(*!
<summary>Checks concrete metadata and name stability across cancellation and Reset for all sixteen tasks.</summary>
<description>Each concrete reset hook is exercised. Cancellation occurs before issuing a native request.</description>
*)
METHOD PROTECTED ExecuteTest
VAR
	expectedTypes : ARRAY [0..15] OF STRING(80) := [
		'CheckDirectoryExists',
		'CreateDirectory',
		'CreateDirectoryIfNotExists',
		'RemoveEmptyDirectory',
		'RemoveEmptyDirectoryIfExists',
		'DeleteFile',
		'RenameFile',
		'LoadFile',
		'FileContentManager',
		'CheckEndOfFile',
		'GetPositionInFile',
		'SetPositionInFile',
		'ReadBytesFromFile',
		'ReadString255FromFile',
		'WriteBytesToFile',
		'WriteString255ToFile'
	];
	expectedName : WSTRING;
	i : DINT;
	caseName : WSTRING;
	started : BOOL;
	cancelled : BOOL;
END_VAR
FOR i := LOWER_BOUND(_Tasks, 1) TO UPPER_BOUND(_Tasks, 1) DO
	caseName := TO_WSTRING(expectedTypes[i]);
	expectedName := TO_WSTRING(TOF_Core.Strings.Concat255(
		expectedTypes[i],
		' (0x',
		Tc2_Utilities.LWORD_TO_HEXSTR(in := TO_LWORD(_Tasks[i].SelfAddress), iPrecision := 16, bLoCase := FALSE),
		')'
	));
	Assert.ThatBool(
		actual := _Tasks[i].Name = expectedName,
		message := TOF_Core.WideStrings.Concat255(caseName, ": Default name must include the concrete type and address")
	).IsTrue();
	Assert.ThatBool(
		actual := _Tasks[i].ClassName = expectedTypes[i],
		message := TOF_Core.WideStrings.Concat255(caseName, ": ", "ClassName must identify the concrete task")
	).IsTrue();
	Assert.ThatBool(
		actual := _Tasks[i].NamespaceName = 'TOF_FileSystem',
		message := TOF_Core.WideStrings.Concat255(caseName, ": ", "Task namespace must identify FileSystem")
	).IsTrue();
	Assert.ThatBool(
		actual := _Tasks[i].State.Ready,
		message := TOF_Core.WideStrings.Concat255(caseName, ": Metadata must leave the task READY")
	).IsTrue();
	started := _Tasks[i].Start();
	Assert.ThatBool(
		actual := started,
		message := TOF_Core.WideStrings.Concat255(caseName, ": ", "Task must accept Start before cancellation")
	).IsTrue();

	IF NOT started THEN
		CONTINUE;
	END_IF

	cancelled := _Tasks[i].Cancel();
	Assert.ThatBool(
		actual := cancelled,
		message := TOF_Core.WideStrings.Concat255(caseName, ": ", "Task must accept Cancel before Execute")
	).IsTrue();

	IF NOT cancelled THEN
		CONTINUE;
	END_IF

	_Tasks[i].Execute();
	Assert.ThatBool(
		actual := _Tasks[i].State.Stopped,
		message := TOF_Core.WideStrings.Concat255(caseName, ": ", "Task must stop after cancellation")
	).IsTrue();
	Assert.ThatBool(
		actual := _Tasks[i].FinalStopReason.ExternalCancel,
		message := TOF_Core.WideStrings.Concat255(caseName, ": ", "Pre-submission cancellation must retain its reason")
	).IsTrue();
	Assert.ThatBool(
		actual := _Tasks[i].Reset(),
		message := TOF_Core.WideStrings.Concat255(caseName, ": ", "Stopped task must accept Reset")
	).IsTrue();
	Assert.ThatBool(
		actual := _Tasks[i].State.Ready,
		message := TOF_Core.WideStrings.Concat255(caseName, ": Reset must restore READY")
	).IsTrue();
	Assert.ThatBool(
		actual := _Tasks[i].Name = expectedName,
		message := TOF_Core.WideStrings.Concat255(caseName, ": Reset must preserve the stored default name")
	).IsTrue();
END_FOR

Assert.ThatBool(
	actual := _ExplicitDirectory.Name = "Explicit directory",
	message := "Directory explicit name must be copied"
).IsTrue();
Assert.ThatBool(
	actual := _ExplicitManager.Name = "Explicit manager",
	message := "Manager explicit name must be copied"
).IsTrue();
Assert.ThatBool(
	actual := _ExplicitRead.Name = "Explicit read",
	message := "Content task explicit name must be copied"
).IsTrue();
END_METHOD

(*!
<summary>Restores the fixtures after a completed or interrupted test.</summary>
<description>
Advances a running task only after cancellation is recorded. Resets fixtures only when they are not already READY.
</description>
*)
METHOD PROTECTED AfterTest
VAR
	i : DINT;
END_VAR
FOR i := LOWER_BOUND(_Tasks, 1) TO UPPER_BOUND(_Tasks, 1) DO
	IF _Tasks[i].State.Running THEN
		IF _Tasks[i].OriginalStopReason.ExternalCancel OR_ELSE _Tasks[i].Cancel() THEN
			_Tasks[i].Execute();
		END_IF
	END_IF

	IF NOT _Tasks[i].State.Ready THEN
		Assert.ThatBool(
			actual := _Tasks[i].Reset(),
			message := TOF_Core.WideStrings.Concat255(_Tasks[i].Name, " must accept Reset during cleanup")
		).IsTrue();
	END_IF
END_FOR
END_METHOD

//! <summary>Borrows the concrete class name for the lifetime of this instance; callers must not modify it.</summary>
{attribute 'monitoring' := 'call'}
PROPERTY ClassName : REFERENCE TO STRING
GET
ClassName REF= _ClassName;
END_GET
END_PROPERTY

//! <summary>Borrows the compiler-initialized namespace; callers must not modify the returned reference.</summary>
{attribute 'monitoring' := 'call'}
PROPERTY NamespaceName : REFERENCE TO STRING
GET
NamespaceName REF= CurrentNamespace.Name;
END_GET
END_PROPERTY

//! <summary>Reports the complete concrete instance size, excluding separately allocated storage.</summary>
{attribute 'monitoring' := 'call'}
PROPERTY SelfSize : ULINT
GET
SelfSize := XSIZEOF(THIS^);
END_GET
END_PROPERTY

END_FUNCTION_BLOCK

// ---- Tests/Files/FileSystemUnboundContentTest.TcPOU
(*
SPDX-FileCopyrightText: © 2026 Oleksandr Tiutyk <trofimich@gmail.com>
SPDX-License-Identifier: MIT
License: https://opensource.org/license/mit
*)

(*!
<summary>Checks all seven unbound content operations and their guarded failure/reset results.</summary>
<description>
The fixture belongs to the runner task and is kept between runs. The test drives no native file requests.
</description>
*)

{attribute 'no_assign'}
{attribute 'no_explicit_call' := 'do not call this function block directly'}
FUNCTION_BLOCK FileSystemUnboundContentTest EXTENDS TOF_Testing.SingleCycleTest
VAR_STAT
	{attribute 'hide'}
	_ClassName : STRING := __POUNAME();
END_VAR
VAR
	_CheckEof : TOF_FileSystem.CheckEndOfFile(name := "unbound CheckEndOfFile");
	_GetPosition : TOF_FileSystem.GetPositionInFile(name := "unbound GetPositionInFile");
	_SetPosition : TOF_FileSystem.SetPositionInFile(name := "unbound SetPositionInFile");
	_ReadBytes : TOF_FileSystem.ReadBytesFromFile(name := "unbound ReadBytesFromFile");
	_ReadString : TOF_FileSystem.ReadString255FromFile(name := "unbound ReadString255FromFile");
	_WriteBytes : TOF_FileSystem.WriteBytesToFile(name := "unbound WriteBytesToFile");
	_WriteString : TOF_FileSystem.WriteString255ToFile(name := "unbound WriteString255ToFile");

	_Tasks : ARRAY [0..6] OF TOF_Tasks.ITask :=
	[
		_CheckEof,
		_GetPosition,
		_SetPosition,
		_ReadBytes,
		_ReadString,
		_WriteBytes,
		_WriteString
	];
END_VAR

(*!
<summary>Checks all seven unbound content operations and their guarded failure/reset results.</summary>
<description>Requires the missing-member diagnostic and checks guarded results in each lifecycle phase.</description>
*)
METHOD PROTECTED ExecuteTest
VAR
	i : DINT;
	message : STRING(255);
	caseName : WSTRING;
	started : BOOL;
END_VAR
checkGuardedResults(phase := "Before Start");

FOR i := LOWER_BOUND(_Tasks, 1) TO UPPER_BOUND(_Tasks, 1) DO
	caseName := _Tasks[i].Name;
	started := _Tasks[i].Start();
	Assert.ThatBool(
		actual := started,
		message := TOF_Core.WideStrings.Concat255(caseName, ": ", "Start must precede validation")
	).IsTrue();

	IF NOT started THEN
		CONTINUE;
	END_IF

	_Tasks[i].Execute();
	_Tasks[i].Execute();
	Assert.ThatBool(
		actual := _Tasks[i].State.Stopped,
		message := TOF_Core.WideStrings.Concat255(caseName, ": ", "Unbound operation must finish failure cleanup")
	).IsTrue();
	Assert.ThatBool(
		actual := _Tasks[i].FinalStopReason.Failure,
		message := TOF_Core.WideStrings.Concat255(caseName, ": ", "Unbound operation must fail")
	).IsTrue();
	message := TO_STRING(_Tasks[i].FinalStopReason.Message);
	Assert.ThatBool(
		actual := TOF_Core.Strings.Contains(
			stringToSearchIn := message,
			stringToFind := '$27FileHandleResource$27'
		),
		message := TOF_Core.WideStrings.Concat255(caseName, ": ", "Unbound failure must identify the missing resource")
	).IsTrue();
END_FOR

checkGuardedResults(phase := "After failure");

FOR i := LOWER_BOUND(_Tasks, 1) TO UPPER_BOUND(_Tasks, 1) DO
	Assert.ThatBool(
		actual := _Tasks[i].Reset(),
		message := TOF_Core.WideStrings.Concat255(_Tasks[i].Name, " must accept Reset")
	).IsTrue();
	Assert.ThatBool(
		actual := _Tasks[i].State.Ready,
		message := TOF_Core.WideStrings.Concat255(_Tasks[i].Name, " must return to READY")
	).IsTrue();
END_FOR

checkGuardedResults(phase := "After Reset");
END_METHOD

(*!
<summary>Checks result defaults when no successful file operation is available.</summary>
<param name="phase">Identifies the observed lifecycle phase in assertion messages.</param>
*)
METHOD PRIVATE checkGuardedResults
VAR_INPUT
	phase : WSTRING;
END_VAR
Assert.ThatBool(
	actual := _CheckEof.IsEndOfFile,
	message := TOF_Core.WideStrings.Concat255(phase, ": CheckEndOfFile.IsEndOfFile")
).IsFalse();
Assert.ThatBool(
	actual := _GetPosition.Position = TOF_Core.SignedInt32.ZERO,
	message := TOF_Core.WideStrings.Concat255(phase, ": ", "Unsuccessful tell must expose zero")
).IsTrue();
Assert.ThatBool(
	actual := _ReadBytes.ActuallyReadBytes = TOF_Core.UnsignedInt32.ZERO,
	message := TOF_Core.WideStrings.Concat255(phase, ": ", "Unsuccessful read count must be zero")
).IsTrue();
Assert.ThatBool(
	actual := _ReadBytes.IsEndOfFile,
	message := TOF_Core.WideStrings.Concat255(phase, ": ", "Unsuccessful read must not expose EOF")
).IsFalse();
Assert.ThatBool(
	actual := _ReadString.ReadString = '',
	message := TOF_Core.WideStrings.Concat255(phase, ": ", "Unsuccessful string read must expose an empty buffer")
).IsTrue();
Assert.ThatBool(
	actual := _ReadString.IsEndOfFile,
	message := TOF_Core.WideStrings.Concat255(phase, ": ", "Unsuccessful string read must not expose EOF")
).IsFalse();
Assert.ThatBool(
	actual := _WriteBytes.ActuallyWrittenBytes = TOF_Core.UnsignedInt32.ZERO,
	message := TOF_Core.WideStrings.Concat255(phase, ": ", "Unsuccessful write count must be zero")
).IsTrue();
END_METHOD

(*!
<summary>Restores the fixtures after a completed or interrupted test.</summary>
<description>
Advances a running task only after cancellation is recorded. Resets fixtures only when they are not already READY.
</description>
*)
METHOD PROTECTED AfterTest
VAR
	i : DINT;
END_VAR
FOR i := LOWER_BOUND(_Tasks, 1) TO UPPER_BOUND(_Tasks, 1) DO
	IF _Tasks[i].State.Running THEN
		IF _Tasks[i].OriginalStopReason.ExternalCancel OR_ELSE _Tasks[i].Cancel() THEN
			_Tasks[i].Execute();
		END_IF
	END_IF

	IF NOT _Tasks[i].State.Ready THEN
		Assert.ThatBool(
			actual := _Tasks[i].Reset(),
			message := TOF_Core.WideStrings.Concat255(_Tasks[i].Name, " must accept Reset during cleanup")
		).IsTrue();
	END_IF
END_FOR
END_METHOD

//! <summary>Borrows the concrete class name for the lifetime of this instance; callers must not modify it.</summary>
{attribute 'monitoring' := 'call'}
PROPERTY ClassName : REFERENCE TO STRING
GET
ClassName REF= _ClassName;
END_GET
END_PROPERTY

//! <summary>Borrows the compiler-initialized namespace; callers must not modify the returned reference.</summary>
{attribute 'monitoring' := 'call'}
PROPERTY NamespaceName : REFERENCE TO STRING
GET
NamespaceName REF= CurrentNamespace.Name;
END_GET
END_PROPERTY

//! <summary>Reports the complete concrete instance size, excluding separately allocated storage.</summary>
{attribute 'monitoring' := 'call'}
PROPERTY SelfSize : ULINT
GET
SelfSize := XSIZEOF(THIS^);
END_GET
END_PROPERTY

END_FUNCTION_BLOCK

// ---- Tests/Files/FileSystemLoadBufferTest.TcPOU
(*
SPDX-FileCopyrightText: © 2026 Oleksandr Tiutyk <trofimich@gmail.com>
SPDX-License-Identifier: MIT
License: https://opensource.org/license/mit
*)

(*!
<summary>Checks null/zero load buffers and the corrected TargetBufferSize diagnostic without native I/O.</summary>
<description>
The fixture belongs to the runner task and is kept between runs. The test drives no native file requests.
</description>
*)

{attribute 'no_assign'}
{attribute 'no_explicit_call' := 'do not call this function block directly'}
FUNCTION_BLOCK FileSystemLoadBufferTest EXTENDS TOF_Testing.SingleCycleTest
VAR_STAT
	{attribute 'hide'}
	_ClassName : STRING := __POUNAME();
END_VAR
VAR
	_Load : TOF_FileSystem.LoadFile(name := "load preconditions");
	_Buffer : BYTE;
END_VAR

(*!
<summary>Checks null/zero load buffers and the corrected TargetBufferSize diagnostic without native I/O.</summary>
<description>Checks the buffer guard order and confirms the fixture can be reconfigured before native submission.</description>
*)
METHOD PROTECTED ExecuteTest
VAR
	started : BOOL;
	cancelled : BOOL;
END_VAR
_Buffer := BYTE#16#A5;
_Load.FilePath := 'unused.bin';

IF NOT checkInvalidBuffer(
	targetBuffer := TOF_Core.Memory.NULL_ADDRESS,
	size := 1,
	propertyToken := '$27TargetBuffer$27',
	caseName := "Null buffer"
)
	OR_ELSE NOT checkInvalidBuffer(
		targetBuffer := ADR(_Buffer),
		size := TOF_Core.UnsignedInt32.ZERO,
		propertyToken := '$27TargetBufferSize$27',
		caseName := "Zero buffer size"
	)
	OR_ELSE NOT checkInvalidBuffer(
		targetBuffer := TOF_Core.Memory.NULL_ADDRESS,
		size := TOF_Core.UnsignedInt32.ZERO,
		propertyToken := '$27TargetBuffer$27',
		caseName := "Null buffer and zero size"
	)
THEN
	RETURN;
END_IF

_Load.TargetBuffer := ADR(_Buffer);
_Load.TargetBufferSize := 1;
started := _Load.Start();
Assert.ThatBool(actual := started, message := "Reconfigured load must accept Start").IsTrue();

IF NOT started THEN
	RETURN;
END_IF

cancelled := _Load.Cancel();
Assert.ThatBool(actual := cancelled, message := "Reconfigured load must accept pre-submission cancellation").IsTrue();

IF NOT cancelled THEN
	RETURN;
END_IF

_Load.Execute();
Assert.ThatBool(actual := _Load.State.Stopped, message := "Cancelled load must stop before submission").IsTrue();
Assert.ThatBool(
	actual := _Load.FinalStopReason.ExternalCancel,
	message := "Pre-submission load cancellation must preserve its reason"
).IsTrue();
Assert.ThatUDInt(actual := _Load.LoadedBytesCount, message := "Cancelled load byte count").ToBe(
	expected := TOF_Core.UnsignedInt32.ZERO
);
Assert.ThatByte(actual := _Buffer, message := "Cancelled load must preserve the caller buffer").ToBe(
	expected := BYTE#16#A5
);
END_METHOD

(*!
<summary>Checks one invalid buffer configuration and resets the stopped task.</summary>
<description>
The reason must identify the exact rejected member before any native request. The caller buffer keeps its sentinel.
Returns TRUE only after the task has accepted Reset and is READY for the next configuration.
</description>
<param name="targetBuffer">Buffer address to pass to LoadFile.</param>
<param name="size">Configured buffer size in bytes.</param>
<param name="propertyToken">Expected member name including the diagnostic quotes.</param>
<param name="caseName">Identifies the buffer configuration in the assertion messages.</param>
*)
METHOD PRIVATE checkInvalidBuffer : BOOL
VAR_INPUT
	targetBuffer : POINTER TO BYTE;
	size : UDINT;
	propertyToken : STRING(32);
	caseName : WSTRING;
END_VAR
VAR
	started : BOOL;
	message : STRING(255);
	resetAccepted : BOOL;
END_VAR
_Load.TargetBuffer := targetBuffer;
_Load.TargetBufferSize := size;
started := _Load.Start();
Assert.ThatBool(
	actual := started,
	message := TOF_Core.WideStrings.Concat255(caseName, ": Start must precede buffer validation")
).IsTrue();

IF NOT started THEN
	RETURN;
END_IF

_Load.Execute();
_Load.Execute();
Assert.ThatBool(
	actual := _Load.State.Stopped,
	message := TOF_Core.WideStrings.Concat255(caseName, ": must finish stopping")
).IsTrue();
Assert.ThatBool(
	actual := _Load.FinalStopReason.Failure,
	message := TOF_Core.WideStrings.Concat255(caseName, ": must fail")
).IsTrue();
message := TO_STRING(_Load.FinalStopReason.Message);
Assert.ThatBool(
	actual := TOF_Core.Strings.Contains(stringToSearchIn := message, stringToFind := propertyToken),
	message := TOF_Core.WideStrings.Concat255(caseName, ": expected diagnostic for ", TO_WSTRING(propertyToken))
).IsTrue();
Assert.ThatUDInt(
	actual := _Load.LoadedBytesCount,
	message := TOF_Core.WideStrings.Concat255(caseName, ": loaded byte count")
).ToBe(expected := TOF_Core.UnsignedInt32.ZERO);
Assert.ThatByte(
	actual := _Buffer,
	message := TOF_Core.WideStrings.Concat255(caseName, ": caller buffer sentinel")
).ToBe(expected := BYTE#16#A5);

resetAccepted := _Load.Reset();
Assert.ThatBool(
	actual := resetAccepted,
	message := TOF_Core.WideStrings.Concat255(caseName, ": must accept Reset")
).IsTrue();
Assert.ThatBool(
	actual := _Load.State.Ready,
	message := TOF_Core.WideStrings.Concat255(caseName, ": Reset must restore READY")
).IsTrue();
checkInvalidBuffer := resetAccepted AND_THEN _Load.State.Ready;
END_METHOD

(*!
<summary>Resets the load task after cancellation, including after an interrupted assertion sequence.</summary>
<description>
Advances a running task only on its cancellation path and reports a task that cannot be reset.
</description>
*)
METHOD PROTECTED AfterTest
IF _Load.State.Running THEN
	IF _Load.OriginalStopReason.ExternalCancel OR_ELSE _Load.Cancel() THEN
		_Load.Execute();
	END_IF
END_IF

Assert.ThatBool(
	actual := _Load.Reset(),
	message := "Load task must be ready after cleanup"
).IsTrue();
END_METHOD

//! <summary>Borrows the concrete class name for the lifetime of this instance; callers must not modify it.</summary>
{attribute 'monitoring' := 'call'}
PROPERTY ClassName : REFERENCE TO STRING
GET
ClassName REF= _ClassName;
END_GET
END_PROPERTY

//! <summary>Borrows the compiler-initialized namespace; callers must not modify the returned reference.</summary>
{attribute 'monitoring' := 'call'}
PROPERTY NamespaceName : REFERENCE TO STRING
GET
NamespaceName REF= CurrentNamespace.Name;
END_GET
END_PROPERTY

//! <summary>Reports the complete concrete instance size, excluding separately allocated storage.</summary>
{attribute 'monitoring' := 'call'}
PROPERTY SelfSize : ULINT
GET
SelfSize := XSIZEOF(THIS^);
END_GET
END_PROPERTY

END_FUNCTION_BLOCK

// ---- Tests/Files/FileSystemQueueBindingTest.TcPOU
(*
SPDX-FileCopyrightText: © 2026 Oleksandr Tiutyk <trofimich@gmail.com>
SPDX-License-Identifier: MIT
License: https://opensource.org/license/mit
*)

(*!
<summary>Checks null enqueue, borrowed binding and READY/RUNNING/STOPPED rebinding rules without opening a file.</summary>
<description>
The fixture belongs to the runner task and is kept between runs. The test drives no native file requests.
</description>
*)

{attribute 'no_assign'}
{attribute 'no_explicit_call' := 'do not call this function block directly'}
FUNCTION_BLOCK FileSystemQueueBindingTest EXTENDS TOF_Testing.SingleCycleTest
VAR_STAT
	{attribute 'hide'}
	_ClassName : STRING := __POUNAME();
END_VAR
VAR CONSTANT
	//! <summary>First path exposed to the child after binding.</summary>
	_InitialFilePath : STRING(255) := 'initial-binding.bin';
	//! <summary>Replacement path used to verify that the child still borrows the resource.</summary>
	_UpdatedFilePath : STRING(255) := 'updated-binding.bin';
END_VAR
VAR
	_Manager : TOF_FileSystem.FileContentManager(name := "binding manager");
	_Read : TOF_FileSystem.ReadBytesFromFile(name := "bound read");
	_Unbound : TOF_FileSystem.ReadBytesFromFile(name := "unbound view");
END_VAR

(*!
<summary>Checks queue membership, the live borrowed binding and state-dependent rebinding without opening a file.</summary>
<description>
The child is removed from the queue before it is driven directly, then cancelled before Execute can submit I/O.
Rejected changes in RUNNING and STOPPED must preserve the existing binding.
</description>
*)
METHOD PROTECTED ExecuteTest
VAR
	exceptionCode : __SYSTEM.ExceptionCode;
	caught : TOF_Core.IException;
	missingArgument : TOF_Core.IArgumentNotSpecifiedException;
	thrown : BOOL;
	started : BOOL;
	cancelled : BOOL;
END_VAR
__TRY
	_Manager.Enqueue(fileHandleTask := 0);
__CATCH(exceptionCode)
	thrown := TRUE;
	caught := TOF_Core.ExceptionManager.GetLastException(
		exceptionCode := exceptionCode,
		catchPointNamespaceName := NamespaceName,
		catchPointPOUName := __POUNAME(),
		catchPointPosition := __POSITION()
	);
	Assert.ThatBool(
		actual := __QUERYINTERFACE(caught, missingArgument),
		message := "Null enqueue must raise ArgumentNotSpecified"
	).IsTrue();
__ENDTRY

Assert.ThatBool(actual := thrown, message := "Null enqueue must raise an exception").IsTrue();
Assert.ThatDInt(actual := _Manager.PendingTaskCount, message := "Null enqueue must leave the queue empty").ToBe(
	expected := 0
);

_Manager.FilePath := _InitialFilePath;
_Manager.Enqueue(fileHandleTask := _Read);
Assert.ThatDInt(actual := _Manager.PendingTaskCount, message := "Enqueue must add the child").ToBe(expected := 1);
Assert.ThatString(
	actual := _Read.FilePath,
	message := "Enqueue must expose the manager's configured file path through the child"
).ToBe(expected := _InitialFilePath);

_Manager.ClearWaitingTasks();
Assert.ThatDInt(actual := _Manager.PendingTaskCount, message := "ClearWaitingTasks must remove the child").ToBe(
	expected := 0
);

IF _Manager.PendingTaskCount <> 0 THEN
	RETURN;
END_IF

_Manager.FilePath := _UpdatedFilePath;
Assert.ThatString(
	actual := _Read.FilePath,
	message := "A removed child must retain a live view of the manager's resource"
).ToBe(expected := _UpdatedFilePath);

Assert.ThatBool(actual := _Read.Reset(), message := "READY Reset is allowed").IsTrue();
Assert.ThatString(
	actual := _Read.FilePath,
	message := "READY Reset must preserve the live binding"
).ToBe(expected := _UpdatedFilePath);

_Read.SetFileHandleResource(fileHandleResource := _Unbound.FileHandleResource);
Assert.ThatBool(
	actual := __ISVALIDREF(_Read.FileHandleResource),
	message := "Invalid resource view must clear a READY binding"
).IsFalse();

_Manager.Enqueue(fileHandleTask := _Read);
_Manager.ClearWaitingTasks();
Assert.ThatDInt(actual := _Manager.PendingTaskCount, message := "Child must be unqueued before direct Start").ToBe(
	expected := 0
);

IF _Manager.PendingTaskCount <> 0 THEN
	RETURN;
END_IF

started := _Read.Start();
Assert.ThatBool(actual := started, message := "Prepared child must accept Start").IsTrue();

IF NOT started THEN
	RETURN;
END_IF

checkRebindingRejected(phase := "RUNNING");

cancelled := _Read.Cancel();
Assert.ThatBool(actual := cancelled, message := "Prepared child must accept pre-submission cancellation").IsTrue();

IF NOT cancelled THEN
	RETURN;
END_IF

_Read.Execute();
Assert.ThatBool(actual := _Read.State.Stopped, message := "Cancelled child must reach STOPPED").IsTrue();

IF NOT _Read.State.Stopped THEN
	RETURN;
END_IF

checkRebindingRejected(phase := "STOPPED");
Assert.ThatBool(actual := _Read.Reset(), message := "Cancelled child must accept Reset").IsTrue();
Assert.ThatBool(
	actual := __ISVALIDREF(_Read.FileHandleResource),
	message := "STOPPED Reset must clear the resource binding"
).IsFalse();
END_METHOD

(*!
<summary>Checks that clearing outside READY raises StandardException and preserves the bound file path.</summary>
<param name="phase">Identifies the child lifecycle phase in assertion messages.</param>
*)
METHOD PRIVATE checkRebindingRejected
VAR_INPUT
	phase : WSTRING;
END_VAR
VAR
	exceptionCode : __SYSTEM.ExceptionCode;
	caught : TOF_Core.IException;
	standard : TOF_Core.IStandardException;
	thrown : BOOL;
END_VAR
__TRY
	_Read.SetFileHandleResource(fileHandleResource := _Unbound.FileHandleResource);
__CATCH(exceptionCode)
	thrown := TRUE;
	caught := TOF_Core.ExceptionManager.GetLastException(
		exceptionCode := exceptionCode,
		catchPointNamespaceName := NamespaceName,
		catchPointPOUName := __POUNAME(),
		catchPointPosition := __POSITION()
	);
	Assert.ThatBool(
		actual := __QUERYINTERFACE(caught, standard),
		message := TOF_Core.WideStrings.Concat255(phase, " rebinding must raise StandardException")
	).IsTrue();
__ENDTRY

Assert.ThatBool(
	actual := thrown,
	message := TOF_Core.WideStrings.Concat255(phase, " rebinding must be rejected")
).IsTrue();
Assert.ThatString(
	actual := _Read.FilePath,
	message := TOF_Core.WideStrings.Concat255(phase, " rebinding refusal must preserve the bound file path")
).ToBe(expected := _UpdatedFilePath);
END_METHOD

(*!
<summary>Removes any waiting child and restores the read fixture.</summary>
<description>
The manager is never started. Teardown can clear the borrowed binding after the child returns to READY.
</description>
*)
METHOD PROTECTED AfterTest
_Manager.ClearWaitingTasks();

IF _Read.State.Running THEN
	IF _Read.OriginalStopReason.ExternalCancel OR_ELSE _Read.Cancel() THEN
		_Read.Execute();
	END_IF
END_IF

Assert.ThatBool(
	actual := _Read.Reset(),
	message := "Read task must be ready after cleanup"
).IsTrue();

IF _Read.State.Ready AND_THEN __ISVALIDREF(_Read.FileHandleResource) THEN
	_Read.SetFileHandleResource(fileHandleResource := _Unbound.FileHandleResource);
END_IF
END_METHOD

//! <summary>Borrows the concrete class name for the lifetime of this instance; callers must not modify it.</summary>
{attribute 'monitoring' := 'call'}
PROPERTY ClassName : REFERENCE TO STRING
GET
ClassName REF= _ClassName;
END_GET
END_PROPERTY

//! <summary>Borrows the compiler-initialized namespace; callers must not modify the returned reference.</summary>
{attribute 'monitoring' := 'call'}
PROPERTY NamespaceName : REFERENCE TO STRING
GET
NamespaceName REF= CurrentNamespace.Name;
END_GET
END_PROPERTY

//! <summary>Reports the complete concrete instance size, excluding separately allocated storage.</summary>
{attribute 'monitoring' := 'call'}
PROPERTY SelfSize : ULINT
GET
SelfSize := XSIZEOF(THIS^);
END_GET
END_PROPERTY

END_FUNCTION_BLOCK

// ---- Tests/Files/FileSystemExceptionCloneTest.TcPOU
(*
SPDX-FileCopyrightText: © 2026 Oleksandr Tiutyk <trofimich@gmail.com>
SPDX-License-Identifier: MIT
License: https://opensource.org/license/mit
*)

(*!
<summary>Checks concrete filesystem exception clones and complete copied diagnostics within one task call.</summary>
<description>
Verifies the concrete exception interfaces and payloads, including a message longer than 255 characters.
Clone references are used only within one test call. The hosting AutomationRunner owns task memory cleanup.
</description>
*)

{attribute 'no_assign'}
{attribute 'no_explicit_call' := 'do not call this function block directly'}
FUNCTION_BLOCK FileSystemExceptionCloneTest EXTENDS TOF_Testing.SingleCycleTest
VAR_STAT
	{attribute 'hide'}
	_ClassName : STRING := __POUNAME();
END_VAR
VAR
	_FileTemplate : TOF_FileSystem.FileSystemException;
	_PathTemplate : TOF_FileSystem.InvalidPathException;
END_VAR

(*!
<summary>Checks concrete filesystem exception clones and complete copied diagnostics within one task call.</summary>
<description>
The filesystem payload crosses the 255-character boundary. Both snapshots must retain their data after
the caller-owned template is cleared. References remain local to the test call.
</description>
*)
METHOD PROTECTED ExecuteTest
VAR
	i : DINT;
	exceptionCode : __SYSTEM.ExceptionCode;
	caught : TOF_Core.IException;
	caughtFile : TOF_FileSystem.IFileSystemException;
	caughtPath : TOF_FileSystem.IInvalidPathException;
	cloned : TOF_Core.IObject;
	fileClone : TOF_FileSystem.IFileSystemException;
	pathClone : TOF_FileSystem.IInvalidPathException;
	message : TOF_Core.ERROR_MESSAGE;
	sourceLocalTimestamp : LDATE_AND_TIME;
	sourceUtcTimestamp : LDATE_AND_TIME;
	path : STRING(255) := 'C:\invalid|path';
	thrown : BOOL;
END_VAR
message := "Native filesystem failure payload: ";

FOR i := 1 TO 5 DO
	TOF_Core.WideStrings.Append255(
		message,
		"Long diagnostic fragment preserving data beyond the 255-character string boundary. "
	);
END_FOR

TOF_Core.WideStrings.Append255(message, "Payload suffix");
Assert.ThatBool(
	actual := TOF_Core.WideStrings.GetLength(value := message) > 255,
	message := "Filesystem clone test payload must exceed 255 characters"
).IsTrue();

__TRY
	_FileTemplate.Throw(
		sourceNamespaceName := 'Tests',
		sourceClassName := 'FileSystemContractTest',
		sourcePOUName := 'FileFailure',
		sourcePosition := 'PositionA',
		message := message,
		errorCode := UDINT#16#70C
	);
__CATCH(exceptionCode)
	thrown := TRUE;
	caught := TOF_Core.ExceptionManager.GetLastException(
		exceptionCode := exceptionCode,
		catchPointNamespaceName := NamespaceName,
		catchPointPOUName := __POUNAME(),
		catchPointPosition := __POSITION()
	);
	Assert.ThatBool(
		actual := __QUERYINTERFACE(caught, caughtFile),
		message := "Throw must retain the concrete filesystem exception"
	).IsTrue();
__ENDTRY

Assert.ThatBool(actual := thrown, message := "Filesystem Throw must propagate").IsTrue();
sourceLocalTimestamp := _FileTemplate.LocalTimestamp;
sourceUtcTimestamp := _FileTemplate.UtcTimestamp;
cloned := _FileTemplate.Clone();
_FileTemplate.Clear();
Assert.ThatBool(
	actual := __QUERYINTERFACE(cloned, fileClone),
	message := "Clone must implement IFileSystemException"
).IsTrue();

IF fileClone <> 0 THEN
	Assert.ThatBool(
		actual := fileClone.IsDynamicInstance,
		message := "Clone must be a dynamic task-owned instance"
	).IsTrue();
	Assert.ThatBool(
		actual := fileClone.SelfAddress <> _FileTemplate.SelfAddress,
		message := "Clone must be distinct from its template"
	).IsTrue();
	Assert.ThatBool(
		actual := fileClone.SourceMessage = message,
		message := "Clone must preserve message payload"
	).IsTrue();
	Assert.ThatBool(
		actual := fileClone.ErrorCode = UDINT#16#70C,
		message := "Clone must preserve native error code"
	).IsTrue();
	Assert.ThatBool(
		actual := fileClone.SourceFullPOUName = 'Tests.FileSystemContractTest.FileFailure()',
		message := "Clone must preserve source POU"
	).IsTrue();
	Assert.ThatBool(
		actual := fileClone.SourcePosition = 'PositionA',
		message := "Clone must preserve source position"
	).IsTrue();
	Assert.ThatBool(
		actual := fileClone.LocalTimestamp = sourceLocalTimestamp,
		message := "Clone must preserve local timestamp"
	).IsTrue();
	Assert.ThatBool(
		actual := fileClone.UtcTimestamp = sourceUtcTimestamp,
		message := "Clone must preserve UTC timestamp"
	).IsTrue();
END_IF

thrown := FALSE;

__TRY
	_PathTemplate.Throw(
		sourceNamespaceName := 'Tests',
		sourceClassName := 'FileSystemContractTest',
		sourcePOUName := 'PathFailure',
		sourcePosition := 'PositionB',
		path := path,
		errorMessage := "Forbidden character"
	);
__CATCH(exceptionCode)
	thrown := TRUE;
	caught := TOF_Core.ExceptionManager.GetLastException(
		exceptionCode := exceptionCode,
		catchPointNamespaceName := NamespaceName,
		catchPointPOUName := __POUNAME(),
		catchPointPosition := __POSITION()
	);
	Assert.ThatBool(
		actual := __QUERYINTERFACE(caught, caughtPath),
		message := "Throw must retain the concrete invalid-path exception"
	).IsTrue();
__ENDTRY

Assert.ThatBool(actual := thrown, message := "Invalid-path Throw must propagate").IsTrue();
sourceLocalTimestamp := _PathTemplate.LocalTimestamp;
sourceUtcTimestamp := _PathTemplate.UtcTimestamp;
cloned := _PathTemplate.Clone();
_PathTemplate.Clear();
Assert.ThatBool(
	actual := __QUERYINTERFACE(cloned, pathClone),
	message := "Clone must implement IInvalidPathException"
).IsTrue();

IF pathClone <> 0 THEN
	Assert.ThatBool(
		actual := pathClone.IsDynamicInstance,
		message := "Path clone must be a dynamic task-owned instance"
	).IsTrue();
	Assert.ThatBool(
		actual := pathClone.SelfAddress <> _PathTemplate.SelfAddress,
		message := "Path clone must be distinct from its template"
	).IsTrue();
	Assert.ThatBool(
		actual := pathClone.SourceMessage = TO_WSTRING('Invalid path $22C:\invalid|path$22: Forbidden character'),
		message := "Path clone must preserve the rejected path and the explanation"
	).IsTrue();
	Assert.ThatBool(
		actual := pathClone.ErrorCode = TOF_Core.UnsignedInt32.ZERO,
		message := "Path clone must preserve error code"
	).IsTrue();
	Assert.ThatBool(
		actual := pathClone.SourceFullPOUName = 'Tests.FileSystemContractTest.PathFailure()',
		message := "Path clone must preserve source POU"
	).IsTrue();
	Assert.ThatBool(
		actual := pathClone.SourcePosition = 'PositionB',
		message := "Path clone must preserve source position"
	).IsTrue();
	Assert.ThatBool(
		actual := pathClone.LocalTimestamp = sourceLocalTimestamp,
		message := "Path clone must preserve local timestamp"
	).IsTrue();
	Assert.ThatBool(
		actual := pathClone.UtcTimestamp = sourceUtcTimestamp,
		message := "Path clone must preserve UTC timestamp"
	).IsTrue();
END_IF
END_METHOD

//! <summary>Borrows the concrete class name for the lifetime of this instance; callers must not modify it.</summary>
{attribute 'monitoring' := 'call'}
PROPERTY ClassName : REFERENCE TO STRING
GET
ClassName REF= _ClassName;
END_GET
END_PROPERTY

//! <summary>Borrows the compiler-initialized namespace; callers must not modify the returned reference.</summary>
{attribute 'monitoring' := 'call'}
PROPERTY NamespaceName : REFERENCE TO STRING
GET
NamespaceName REF= CurrentNamespace.Name;
END_GET
END_PROPERTY

//! <summary>Reports the complete concrete instance size, excluding separately allocated storage.</summary>
{attribute 'monitoring' := 'call'}
PROPERTY SelfSize : ULINT
GET
SelfSize := XSIZEOF(THIS^);
END_GET
END_PROPERTY

END_FUNCTION_BLOCK

// ---- Tests/Files/FileSystemManagerStartRefusalTest.TcPOU
(*
SPDX-FileCopyrightText: © 2026 Oleksandr Tiutyk <trofimich@gmail.com>
SPDX-License-Identifier: MIT
License: https://opensource.org/license/mit
*)

(*!
<summary>Checks that a manager can retry Start directly after a contained preparation failure.</summary>
<description>
The fixture belongs to the runner task and is kept between runs. The test drives no native file requests.
</description>
*)

{attribute 'no_assign'}
{attribute 'no_explicit_call' := 'do not call this function block directly'}
FUNCTION_BLOCK FileSystemManagerStartRefusalTest EXTENDS TOF_Testing.SingleCycleTest
VAR_STAT
	{attribute 'hide'}
	_ClassName : STRING := __POUNAME();
END_VAR
VAR
	_Manager : FileManagerStartRefusalProbe(name := "refused file manager");
END_VAR

(*!
<summary>Checks that a refused start leaves the manager idle and eligible for an immediate successful retry.</summary>
<description>Disables the injected refusal and cancels the accepted retry before advancing acquisition.</description>
*)
METHOD PROTECTED ExecuteTest
VAR
	accepted : BOOL;
	cancelled : BOOL;
	refuseReason : TOF_Core.ERROR_MESSAGE;
	refuseText : STRING(255);
END_VAR
_Manager.FilePath := 'unused.bin';
_Manager.RefuseStart := TRUE;
accepted := _Manager.Start(refuseReason => refuseReason);
refuseText := TO_STRING(refuseReason);
Assert.ThatBool(actual := accepted, message := "Preparation exception must refuse Start").IsFalse();
Assert.ThatBool(actual := _Manager.State.Ready, message := "Refused Start must leave the manager READY").IsTrue();
Assert.ThatBool(
	actual := TOF_Core.Strings.Contains(
		stringToSearchIn := refuseText,
		stringToFind := 'Synthetic file-manager Start refusal'
	),
	message := "Refused Start must identify the preparation failure"
).IsTrue();
Assert.ThatBool(
	actual := _Manager.ResourceManager.ResourceAcquired,
	message := "Refused Start must acquire no resource"
).IsFalse();

IF accepted OR_ELSE NOT _Manager.State.Ready THEN
	RETURN;
END_IF

_Manager.Execute();
Assert.ThatBool(
	actual := _Manager.State.Ready,
	message := "Execute after refusal must not initiate acquisition"
).IsTrue();
Assert.ThatBool(
	actual := _Manager.ResourceManager.ResourceAcquired,
	message := "Execute after refusal must leave the resource unacquired"
).IsFalse();

IF NOT _Manager.State.Ready THEN
	RETURN;
END_IF

_Manager.RefuseStart := FALSE;
accepted := _Manager.Start();
Assert.ThatBool(actual := accepted, message := "Start must allow a retry without Reset").IsTrue();

IF NOT accepted THEN
	RETURN;
END_IF

cancelled := _Manager.Cancel();
Assert.ThatBool(actual := cancelled, message := "Cancel must be accepted before file acquisition").IsTrue();

IF NOT cancelled THEN
	RETURN;
END_IF

_Manager.Execute();
Assert.ThatBool(actual := _Manager.State.Stopped, message := "Cancelled retry must reach STOPPED").IsTrue();
Assert.ThatBool(
	actual := _Manager.FinalStopReason.ExternalCancel,
	message := "The successful retry must report its own cancellation"
).IsTrue();
END_METHOD

(*!
<summary>Cancels an unexpectedly started manager before advancing it and resets the fixture.</summary>
*)
METHOD PROTECTED AfterTest
IF _Manager.State.Running THEN
	IF _Manager.OriginalStopReason.ExternalCancel OR_ELSE _Manager.Cancel() THEN
		_Manager.Execute();
	END_IF
END_IF

Assert.ThatBool(
	actual := _Manager.Reset(),
	message := "File manager must be ready after cleanup"
).IsTrue();
END_METHOD

//! <summary>Borrows the concrete class name for the lifetime of this instance; callers must not modify it.</summary>
{attribute 'monitoring' := 'call'}
PROPERTY ClassName : REFERENCE TO STRING
GET
ClassName REF= _ClassName;
END_GET
END_PROPERTY

//! <summary>Borrows the compiler-initialized namespace; callers must not modify the returned reference.</summary>
{attribute 'monitoring' := 'call'}
PROPERTY NamespaceName : REFERENCE TO STRING
GET
NamespaceName REF= CurrentNamespace.Name;
END_GET
END_PROPERTY

//! <summary>Reports the complete concrete instance size, excluding separately allocated storage.</summary>
{attribute 'monitoring' := 'call'}
PROPERTY SelfSize : ULINT
GET
SelfSize := XSIZEOF(THIS^);
END_GET
END_PROPERTY

END_FUNCTION_BLOCK

// ---- Tests/Files/FileManagerStartRefusalProbe.TcPOU
(*
SPDX-FileCopyrightText: © 2026 Oleksandr Tiutyk <trofimich@gmail.com>
SPDX-License-Identifier: MIT
License: https://opensource.org/license/mit
*)

(*!
<summary>Injects a configurable file-manager start preparation exception.</summary>
<description>
Set RefuseStart while READY. With refusal disabled, the probe runs the real file-manager preparation hook.
The test cancels accepted starts before driving native acquisition.
</description>
*)

FUNCTION_BLOCK FileManagerStartRefusalProbe EXTENDS TOF_FileSystem.FileContentManager
VAR_STAT
	_ProbeClassName : STRING := __POUNAME();
END_VAR
VAR_INPUT
	//! <summary>Requests a synthetic preparation exception on the next Start.</summary>
	RefuseStart : BOOL;
END_VAR

(*!
<summary>Raises the requested test exception or delegates to normal file-manager preparation.</summary>
*)
METHOD PROTECTED OnBeforeStart
IF RefuseStart THEN
	TOF_Core.Exceptions.ThrowStandard(
		sourceNamespaceName := NamespaceName,
		sourceClassName := ClassName,
		sourcePOUName := __POUNAME(),
		sourcePosition := __POSITION(),
		message := "Synthetic file-manager Start refusal"
	);
END_IF

SUPER^.OnBeforeStart();
END_METHOD

(*!
<summary>Borrows initialized read-only type metadata without exceptions or resource initialization.</summary>
*)
PROPERTY ClassName : REFERENCE TO STRING
GET
ClassName REF= _ProbeClassName;
END_GET
END_PROPERTY

(*!
<summary>Borrows compiler-initialized read-only metadata identifying the test namespace.</summary>
*)
PROPERTY NamespaceName : REFERENCE TO STRING
GET
NamespaceName REF= CurrentNamespace.Name;
END_GET
END_PROPERTY

(*!
<summary>Reports the size of this concrete probe in bytes.</summary>
*)
PROPERTY SelfSize : ULINT
GET
SelfSize := XSIZEOF(THIS^);
END_GET
END_PROPERTY

END_FUNCTION_BLOCK

// ---- Tests/Files/DirectoryTest.TcPOU
(*
SPDX-FileCopyrightText: © 2026 Oleksandr Tiutyk <trofimich@gmail.com>
SPDX-License-Identifier: MIT
License: https://opensource.org/license/mit
*)

(*!
<summary>Groups the three native directory scenarios.</summary>
<description>
Owns one independent fixture per child and borrows the shared FileTestRoot. Use from one task without reentry.
The child array and parent associations stay fixed. Do not copy the group or modify its borrowed array.
</description>
*)

{attribute 'no_assign'}
{attribute 'no_explicit_call' := 'do not call this function block directly'}
FUNCTION_BLOCK DirectoryTest EXTENDS TOF_Testing.TestGroup<3>
VAR_STAT
	{attribute 'hide'}
	_ClassName : STRING := __POUNAME();
END_VAR
VAR
	_CreateAndRemove : DirectoryOperationTest(
		name := "CheckThenCreateThenRemoveDirectory",
		parent := THIS^,
		directoryPath := 'C:\OpenFrameworkTests\DirectoryTest_CreateRemove',
		firstStep := DIRECTORY_TEST_STEP.CHECK_DIRECTORY_PRESENT
	);
	_MissingChild : DirectoryOperationTest(
		name := "CheckInvalidDirectory",
		parent := THIS^,
		directoryPath := 'C:\OpenFrameworkTests\DirectoryTest_Missing',
		firstStep := DIRECTORY_TEST_STEP.CHECK_CHILD_DIRECTORY_ABSENT
	);
	_ConditionalOperations : DirectoryOperationTest(
		name := "CreateDirectoryIfNotExistsThenRemoveItIfExists",
		parent := THIS^,
		directoryPath := 'C:\OpenFrameworkTests\DirectoryTest_IfExists',
		firstStep := DIRECTORY_TEST_STEP.CREATE_CHILD_DIRECTORY
	);

	_Children : ARRAY [0.._ChildCount - 1] OF TOF_Testing.ITestElement :=
	[
		_CreateAndRemove,
		_MissingChild,
		_ConditionalOperations
	];
END_VAR

//! <summary>Borrows the fixed array of this concrete group; do not modify it.</summary>
{attribute 'monitoring' := 'call'}
PROPERTY Children : REFERENCE TO ARRAY [0.._ChildCount - 1] OF TOF_Testing.ITestElement
GET
Children REF= _Children;
END_GET
END_PROPERTY

//! <summary>Borrows the concrete class name for the lifetime of this instance; callers must not modify it.</summary>
{attribute 'monitoring' := 'call'}
PROPERTY ClassName : REFERENCE TO STRING
GET
ClassName REF= _ClassName;
END_GET
END_PROPERTY

//! <summary>Borrows the compiler-initialized namespace; callers must not modify the returned reference.</summary>
{attribute 'monitoring' := 'call'}
PROPERTY NamespaceName : REFERENCE TO STRING
GET
NamespaceName REF= CurrentNamespace.Name;
END_GET
END_PROPERTY

//! <summary>Reports the complete concrete instance size, excluding separately allocated storage.</summary>
{attribute 'monitoring' := 'call'}
PROPERTY SelfSize : ULINT
GET
SelfSize := XSIZEOF(THIS^);
END_GET
END_PROPERTY

END_FUNCTION_BLOCK

// ---- Tests/Files/DirectoryOperationTest.TcPOU
(*
SPDX-FileCopyrightText: © 2026 Oleksandr Tiutyk <trofimich@gmail.com>
SPDX-License-Identifier: MIT
License: https://opensource.org/license/mit
*)

(*!
<summary>Runs one native directory lifecycle scenario.</summary>
<description>
The caller reserves a fixed directory under FileTestRoot and drives this leaf in one task without reentry.
Ordinary creation establishes ownership. A refusal, collision or interrupted create grants no ownership.
The scenario retains ownership until a successful existence query confirms removal. Pending operations
are drained and owned paths are removed nonrecursively before reporting. A failed cleanup can require
inspection before reuse. The scenario deadline includes root preparation. Do not copy the instance.
</description>
*)

{attribute 'no_assign'}
{attribute 'no_explicit_call' := 'do not call this function block directly'}
FUNCTION_BLOCK DirectoryOperationTest EXTENDS TOF_Testing.MultiCycleTest
VAR_STAT
	{attribute 'hide'}
	_ClassName : STRING := __POUNAME();
END_VAR
VAR CONSTANT
	//! <summary>Timeout passed to each native directory operation.</summary>
	_NativeTimeout : TIME := T#2S;
	//! <summary>Time allowed for preparation and work before requesting cleanup.</summary>
	_ScenarioTimeout : TIME := T#10S;
END_VAR
VAR
	_DirectoryPath : STRING(255);
	_ChildPath : STRING(255);
	_FirstStep : DIRECTORY_TEST_STEP;
	_Step : DIRECTORY_TEST_STEP;
	_Lifecycle : FILE_TEST_LIFECYCLE;
	_ScenarioDeadline : Tc2_Standard.TON;
	_ActiveOperation : TOF_Tasks.ITask;
	_OwnsDirectory : BOOL;
	_OwnsChildDirectory : BOOL;
	_ChildCleanupFinished : BOOL;
	_ScenarioFailure : TOF_Core.ERROR_MESSAGE;
	_CleanupFailure : TOF_Core.ERROR_MESSAGE;

	_CreateDirectory : TOF_FileSystem.CreateDirectory(name := "CreateDirectory");
	_CheckDirectory : TOF_FileSystem.CheckDirectoryExists(name := "CheckDirectoryExists");
	_RemoveDirectory : TOF_FileSystem.RemoveEmptyDirectory(name := "RemoveEmptyDirectory");
	_CreateChild : TOF_FileSystem.CreateDirectoryIfNotExists(name := "CreateDirectoryIfNotExists");
	_RemoveChild : TOF_FileSystem.RemoveEmptyDirectoryIfExists(name := "RemoveEmptyDirectoryIfExists");
	_CleanupChild : TOF_FileSystem.RemoveEmptyDirectoryIfExists(name := "Remove owned child directory");
	_CleanupDirectory : TOF_FileSystem.RemoveEmptyDirectoryIfExists(name := "Remove owned scenario directory");
END_VAR

(*!
<summary>Stores the fixed scenario path and selects its first check after creation.</summary>
<description>
Initialization performs no I/O. The inherited initializer stores name and parent. Use CHECK_DIRECTORY_PRESENT,
CHECK_CHILD_DIRECTORY_ABSENT or CREATE_CHILD_DIRECTORY for firstStep. The scenario deadline excludes cleanup.
</description>
<param name="name">Name used in the test report.</param>
<param name="parent">Group that owns this test.</param>
<param name="directoryPath">Reserved scenario path below the shared filesystem test root.</param>
<param name="firstStep">First step after ordinary creation.</param>
*)
METHOD FB_init : BOOL
VAR_INPUT
	bInitRetains: BOOL; // TRUE: the retain variables are initialized (reset warm / reset cold)
	bInCopyCode: BOOL; // TRUE: the instance will be copied to the copy code afterward (online change)
	name : WSTRING;
	parent : TOF_Testing.ITestElement;
	directoryPath : STRING(255);
	firstStep : DIRECTORY_TEST_STEP;
END_VAR
_DirectoryPath := directoryPath;
_FirstStep := firstStep;

// Keep the test alive while cyclic cleanup is pending after the scenario deadline.
_Timeout := T#0S;
FB_init := TRUE;
END_METHOD

(*!
<summary>Rearms the directory fixture without submitting native operations.</summary>
<description>
Unresolved ownership or pending operations from a previous run fail this leaf before another path is touched.
</description>
*)
METHOD PROTECTED BeforeTest
IF _ActiveOperation <> 0 OR_ELSE _OwnsDirectory OR_ELSE _OwnsChildDirectory THEN
	RecordFailure(message := "The previous run left unresolved directory ownership or a pending task");
	RETURN;
END_IF

IF NOT _CleanupChild.Reset() OR_ELSE NOT _CleanupDirectory.Reset() THEN
	RecordFailure(message := "Directory cleanup tasks refused Reset");
	RETURN;
END_IF

_ChildPath := TOF_Core.Strings.Concat255(_DirectoryPath, '\Child');
_CreateDirectory.DirectoryPath := _DirectoryPath;
_RemoveDirectory.DirectoryPath := _DirectoryPath;
_CreateChild.DirectoryPath := _ChildPath;
_RemoveChild.DirectoryPath := _ChildPath;
_CleanupChild.DirectoryPath := _ChildPath;
_CleanupDirectory.DirectoryPath := _DirectoryPath;

_CreateDirectory.Timeout := _NativeTimeout;
_CheckDirectory.Timeout := _NativeTimeout;
_RemoveDirectory.Timeout := _NativeTimeout;
_CreateChild.Timeout := _NativeTimeout;
_RemoveChild.Timeout := _NativeTimeout;
_CleanupChild.Timeout := _NativeTimeout;
_CleanupDirectory.Timeout := _NativeTimeout;

_CreateDirectory.PathType := Tc2_System.E_OpenPath.PATH_GENERIC;
_CheckDirectory.PathType := Tc2_System.E_OpenPath.PATH_GENERIC;
_RemoveDirectory.PathType := Tc2_System.E_OpenPath.PATH_GENERIC;
_CreateChild.PathType := Tc2_System.E_OpenPath.PATH_GENERIC;
_RemoveChild.PathType := Tc2_System.E_OpenPath.PATH_GENERIC;
_CleanupChild.PathType := Tc2_System.E_OpenPath.PATH_GENERIC;
_CleanupDirectory.PathType := Tc2_System.E_OpenPath.PATH_GENERIC;

_ScenarioDeadline(IN := FALSE, PT := _ScenarioTimeout);
_ScenarioFailure := "";
_CleanupFailure := "";
_ChildCleanupFinished := FALSE;
_Step := DIRECTORY_TEST_STEP.CREATE_DIRECTORY;
_Lifecycle := FILE_TEST_LIFECYCLE.RUNNING_SCENARIO;
END_METHOD

(*!
<summary>Advances scenario work or cleanup and reports the final outcome.</summary>
<description>
An assertion failure would terminate the leaf immediately. Retain the first scenario failure in instance storage
and publish it with any cleanup diagnostic only after cooperative stopping and removal attempts finish.
</description>
*)
METHOD PROTECTED ExecuteTest : TOF_Testing.TEST_CYCLE_RESULT
ExecuteTest := TOF_Testing.TEST_CYCLE_RESULT.BUSY;

IF _Lifecycle = FILE_TEST_LIFECYCLE.RUNNING_SCENARIO THEN
	__TRY
		runScenario();
	__CATCH
		_ScenarioFailure := "Exception interrupted the directory operation; inspect any unfinished creation";
	__ENDTRY

	IF _ScenarioFailure <> "" OR_ELSE _Step = DIRECTORY_TEST_STEP.COMPLETED THEN
		_Lifecycle := FILE_TEST_LIFECYCLE.CLEANING_UP;
	END_IF

	RETURN;
END_IF

__TRY
	IF NOT runCleanup() THEN
		RETURN;
	END_IF
__CATCH
	IF _CleanupFailure = "" THEN
		_CleanupFailure := "An exception interrupted cleanup; inspect the directory if artifacts remain";
	END_IF

	RETURN;
__ENDTRY

_Lifecycle := FILE_TEST_LIFECYCLE.FINISHED;
ExecuteTest := TOF_Testing.TEST_CYCLE_RESULT.DONE;

IF _ScenarioFailure <> "" OR_ELSE _CleanupFailure <> "" THEN
	reportFailure();
END_IF
END_METHOD

(*!
<summary>Advances one step of the chosen directory scenario.</summary>
<description>
The same deadline covers waiting for the shared root and advancing native operations. A failure is
copied to _ScenarioFailure for later reporting. The conditional scenario also checks native refusal to remove
a nonempty parent and confirms the child survived. Ownership is retained until absence is observed.
</description>
*)
METHOD PRIVATE runScenario
VAR
	removalMessage : STRING(255);
	expectedDiagnostic : STRING(255);
END_VAR
_ScenarioDeadline(IN := TRUE, PT := _ScenarioTimeout);

IF FileTestRoot.FailureMessage <> TOF_Core.Strings.Empty THEN
	_ScenarioFailure := TO_WSTRING(FileTestRoot.FailureMessage);
	RETURN;
END_IF

IF _ScenarioDeadline.Q THEN
	_ScenarioFailure := "Scenario exceeded 10 seconds; inspect any directory whose creation was interrupted";
	RETURN;
END_IF

IF NOT FileTestRoot.Prepared THEN
	RETURN;
END_IF

CASE _Step OF
	DIRECTORY_TEST_STEP.CREATE_DIRECTORY:
		IF advanceOperation(operation := _CreateDirectory) THEN
			_OwnsDirectory := TRUE;
			_Step := _FirstStep;
		END_IF

	DIRECTORY_TEST_STEP.CHECK_DIRECTORY_PRESENT:
		IF verifyDirectory(directoryPath := _DirectoryPath, expectedExists := TRUE) THEN
			_Step := DIRECTORY_TEST_STEP.REMOVE_DIRECTORY;
		END_IF

	DIRECTORY_TEST_STEP.CREATE_CHILD_DIRECTORY:
		IF advanceOperation(operation := _CreateChild) THEN
			_OwnsChildDirectory := TRUE;
			_Step := DIRECTORY_TEST_STEP.CHECK_CHILD_DIRECTORY_PRESENT;
		END_IF

	DIRECTORY_TEST_STEP.CHECK_CHILD_DIRECTORY_PRESENT:
		IF verifyDirectory(directoryPath := _ChildPath, expectedExists := TRUE) THEN
			_Step := DIRECTORY_TEST_STEP.CREATE_CHILD_DIRECTORY_AGAIN;
		END_IF

	DIRECTORY_TEST_STEP.CREATE_CHILD_DIRECTORY_AGAIN:
		IF advanceOperation(operation := _CreateChild) THEN
			_Step := DIRECTORY_TEST_STEP.CHECK_CHILD_DIRECTORY_PRESENT_AGAIN;
		END_IF

	DIRECTORY_TEST_STEP.CHECK_CHILD_DIRECTORY_PRESENT_AGAIN:
		IF verifyDirectory(directoryPath := _ChildPath, expectedExists := TRUE) THEN
			_Step := DIRECTORY_TEST_STEP.REJECT_NONEMPTY_DIRECTORY_REMOVAL;
		END_IF

	DIRECTORY_TEST_STEP.REJECT_NONEMPTY_DIRECTORY_REMOVAL:
		IF advanceOperation(operation := _RemoveDirectory, expectedReason := TOF_Tasks.TASK_STOP_REASON.FAILURE) THEN
			removalMessage := TO_STRING(_RemoveDirectory.FinalStopReason.Message);
			expectedDiagnostic := TOF_Core.Strings.Concat255('while removing directory $27', _DirectoryPath, '$27');

			IF NOT TOF_Core.Strings.Contains(stringToSearchIn := removalMessage, stringToFind := expectedDiagnostic) THEN
				_ScenarioFailure := TOF_Core.WideStrings.ConcatFit255(
					"Expected a native failure removing the nonempty directory: ",
					TO_WSTRING(removalMessage)
				);
			ELSE
				_Step := DIRECTORY_TEST_STEP.CHECK_CHILD_DIRECTORY_RETAINED;
			END_IF
		END_IF

	DIRECTORY_TEST_STEP.CHECK_CHILD_DIRECTORY_RETAINED:
		IF verifyDirectory(directoryPath := _ChildPath, expectedExists := TRUE) THEN
			_Step := DIRECTORY_TEST_STEP.REMOVE_CHILD_DIRECTORY;
		END_IF

	DIRECTORY_TEST_STEP.REMOVE_CHILD_DIRECTORY:
		IF advanceOperation(operation := _RemoveChild) THEN
			_Step := DIRECTORY_TEST_STEP.CHECK_CHILD_DIRECTORY_ABSENT;
		END_IF

	DIRECTORY_TEST_STEP.CHECK_CHILD_DIRECTORY_ABSENT:
		IF verifyDirectory(directoryPath := _ChildPath, expectedExists := FALSE) THEN
			IF _FirstStep = DIRECTORY_TEST_STEP.CHECK_CHILD_DIRECTORY_ABSENT THEN
				_Step := DIRECTORY_TEST_STEP.REMOVE_DIRECTORY;
			ELSE
				_Step := DIRECTORY_TEST_STEP.REMOVE_CHILD_DIRECTORY_AGAIN;
			END_IF
		END_IF

	DIRECTORY_TEST_STEP.REMOVE_CHILD_DIRECTORY_AGAIN:
		IF advanceOperation(operation := _RemoveChild) THEN
			_Step := DIRECTORY_TEST_STEP.CHECK_CHILD_DIRECTORY_ABSENT_AGAIN;
		END_IF

	DIRECTORY_TEST_STEP.CHECK_CHILD_DIRECTORY_ABSENT_AGAIN:
		IF verifyDirectory(directoryPath := _ChildPath, expectedExists := FALSE) THEN
			_OwnsChildDirectory := FALSE;
			_Step := DIRECTORY_TEST_STEP.REMOVE_DIRECTORY;
		END_IF

	DIRECTORY_TEST_STEP.REMOVE_DIRECTORY:
		IF advanceOperation(operation := _RemoveDirectory) THEN
			_Step := DIRECTORY_TEST_STEP.CHECK_DIRECTORY_ABSENT;
		END_IF

	DIRECTORY_TEST_STEP.CHECK_DIRECTORY_ABSENT:
		IF verifyDirectory(directoryPath := _DirectoryPath, expectedExists := FALSE) THEN
			_OwnsDirectory := FALSE;
			_Step := DIRECTORY_TEST_STEP.COMPLETED;
		END_IF

	ELSE
		_ScenarioFailure := "Unexpected directory scenario step";
END_CASE
END_METHOD

(*!
<summary>Starts or advances the specified scenario task for one PLC cycle.</summary>
<description>
Pass the same task and expected reason until the step finishes. TRUE requires STOPPED with the expected final
reason. A refusal or unexpected reason is copied for the test result. Cleanup may cancel the active task.
</description>
<param name="operation">Persistent task belonging to this scenario.</param>
<param name="expectedReason">Final stop reason required to advance to the next verification step.</param>
*)
METHOD PRIVATE advanceOperation : BOOL
VAR_INPUT
	operation : TOF_Tasks.ITask;
	expectedReason : TOF_Tasks.TASK_STOP_REASON := TOF_Tasks.TASK_STOP_REASON.WORK_DONE;
END_VAR
VAR
	operationMessage : TOF_Core.ERROR_MESSAGE;
END_VAR
IF _ActiveOperation = 0 THEN
	_ActiveOperation := operation;

	IF NOT operation.Reset(refuseReason => operationMessage) THEN
		_ScenarioFailure := "Reset refused: ";
		TOF_Core.WideStrings.AppendFit(targetString := _ScenarioFailure, sourceString := operationMessage);
		RETURN;
	END_IF

	IF NOT operation.Start(refuseReason => operationMessage) THEN
		_ScenarioFailure := "Start refused: ";
		TOF_Core.WideStrings.AppendFit(targetString := _ScenarioFailure, sourceString := operationMessage);
		RETURN;
	END_IF
END_IF

operation.Execute();

IF NOT operation.State.Stopped THEN
	RETURN;
END_IF

_ActiveOperation := 0;
advanceOperation := operation.FinalStopReason.Value = expectedReason;

IF NOT advanceOperation THEN
	_ScenarioFailure := TOF_Core.WideStrings.ConcatFit255(
		operation.Name,
		" stopped with ",
		TO_WSTRING(operation.FinalStopReason.Value),
		", expected ",
		TO_WSTRING(expectedReason),
		": "
	);
	operationMessage := operation.FinalStopReason.Message;
	TOF_Core.WideStrings.AppendFit(targetString := _ScenarioFailure, sourceString := operationMessage);
END_IF
END_METHOD

(*!
<summary>Checks the result of a native existence query against the expected state.</summary>
<description>
TRUE requires both a successful native task and a matching observation. Pending queries retain their path.
</description>
<param name="directoryPath">Fixed path to query for this step.</param>
<param name="expectedExists">Required value of DirectoryExists.</param>
*)
METHOD PRIVATE verifyDirectory : BOOL
VAR_INPUT
	directoryPath : STRING(255);
	expectedExists : BOOL;
END_VAR
IF _ActiveOperation = 0 THEN
	_CheckDirectory.DirectoryPath := directoryPath;
END_IF

IF NOT advanceOperation(operation := _CheckDirectory) THEN
	RETURN;
END_IF

verifyDirectory := _CheckDirectory.DirectoryExists = expectedExists;

IF NOT verifyDirectory THEN
	_ScenarioFailure := TOF_Core.WideStrings.ConcatFit255(
		"DirectoryExists expected ", TO_WSTRING(expectedExists), " for ", TO_WSTRING(directoryPath)
	);
END_IF
END_METHOD

(*!
<summary>Drains in-flight work and advances removal of owned directories.</summary>
<description>
Cleanup removes the child before the parent. It never adopts a pre-existing path, uses no recursive
deletion and is allowed to outlive the scenario deadline. TRUE reports finished attempts.
</description>
*)
METHOD PRIVATE runCleanup : BOOL
VAR
	removed : BOOL;
END_VAR
IF FileTestRoot.Running THEN
	RETURN;
END_IF

IF _ActiveOperation <> 0 THEN
	IF _ActiveOperation.State.Running THEN
		IF NOT _ActiveOperation.OriginalStopReason.ExternalCancel THEN
			_ActiveOperation.Cancel();
		END_IF

		_ActiveOperation.Execute();

		IF _ActiveOperation.State.Running THEN
			RETURN;
		END_IF
	END_IF

	_ActiveOperation := 0;
END_IF

IF _OwnsChildDirectory AND_THEN NOT _ChildCleanupFinished THEN
	IF NOT advanceCleanupRemoval(operation := _CleanupChild, removed => removed) THEN
		RETURN;
	END_IF

	_ChildCleanupFinished := TRUE;
	_OwnsChildDirectory := NOT removed;
END_IF

IF _OwnsDirectory THEN
	IF NOT advanceCleanupRemoval(operation := _CleanupDirectory, removed => removed) THEN
		RETURN;
	END_IF

	_OwnsDirectory := NOT removed;
END_IF

runCleanup := TRUE;
END_METHOD

(*!
<summary>Advances one nonrecursive removal and copies its diagnostic.</summary>
<description>
Returns TRUE after a failed Start or a stopped task. If the task is still running, the next cycle advances it.
</description>
<param name="operation">Persistent removal task configured for a path owned by this scenario.</param>
<param name="removed">TRUE only when the removal task stopped with WORK_DONE.</param>
*)
METHOD PRIVATE advanceCleanupRemoval : BOOL
VAR_INPUT
	operation : TOF_Tasks.ITask;
END_VAR
VAR_OUTPUT
	removed : BOOL;
END_VAR
VAR
	failure : TOF_Core.ERROR_MESSAGE;
END_VAR
removed := FALSE;

IF operation.State.Ready AND_THEN NOT operation.Start(refuseReason => failure) THEN
	IF failure = "" THEN
		failure := "Start refused";
	END_IF
ELSE
	operation.Execute();

	IF NOT operation.State.Stopped THEN
		RETURN;
	END_IF

	removed := operation.FinalStopReason.WorkDone;

	IF NOT removed THEN
		failure := operation.FinalStopReason.Message;

		IF failure = "" THEN
			failure := "Stopped without WORK_DONE";
		END_IF
	END_IF
END_IF

IF NOT removed THEN
	IF _CleanupFailure <> "" THEN
		TOF_Core.WideStrings.AppendFit(targetString := _CleanupFailure, sourceString := " | ");
	END_IF

	TOF_Core.WideStrings.AppendFit255(_CleanupFailure, operation.Name, ": ");
	TOF_Core.WideStrings.AppendFit(targetString := _CleanupFailure, sourceString := failure);
END_IF

advanceCleanupRemoval := TRUE;
END_METHOD

(*!
<summary>Reports the failing path and step after cleanup.</summary>
<description>
Preserves the original diagnostic and adds cleanup information within the available result capacity.
</description>
*)
METHOD PRIVATE reportFailure
VAR
	message : TOF_Core.ERROR_MESSAGE;
END_VAR
message := TOF_Core.WideStrings.ConcatFit255(TO_WSTRING(_DirectoryPath), " [", TO_WSTRING(_Step), "]: ");

IF _ScenarioFailure <> "" THEN
	TOF_Core.WideStrings.AppendFit(targetString := message, sourceString := _ScenarioFailure);
END_IF

IF _CleanupFailure <> "" THEN
	IF _ScenarioFailure <> "" THEN
		TOF_Core.WideStrings.AppendFit(targetString := message, sourceString := " | ");
	END_IF

	TOF_Core.WideStrings.AppendFit255(message, "Cleanup: ");
	TOF_Core.WideStrings.AppendFit(targetString := message, sourceString := _CleanupFailure);
END_IF

RecordFailure(message := message);
END_METHOD

//! <summary>Borrows the concrete class name for the lifetime of this instance; callers must not modify it.</summary>
{attribute 'monitoring' := 'call'}
PROPERTY ClassName : REFERENCE TO STRING
GET
ClassName REF= _ClassName;
END_GET
END_PROPERTY

//! <summary>Borrows the compiler-initialized namespace; callers must not modify the returned reference.</summary>
{attribute 'monitoring' := 'call'}
PROPERTY NamespaceName : REFERENCE TO STRING
GET
NamespaceName REF= CurrentNamespace.Name;
END_GET
END_PROPERTY

//! <summary>Reports the complete concrete instance size, excluding separately allocated storage.</summary>
{attribute 'monitoring' := 'call'}
PROPERTY SelfSize : ULINT
GET
SelfSize := XSIZEOF(THIS^);
END_GET
END_PROPERTY

END_FUNCTION_BLOCK

// ---- Tests/Files/FileContentManagerOperationsTest.TcPOU
(*
SPDX-FileCopyrightText: c 2026 Oleksandr Tiutyk <trofimich@gmail.com>
SPDX-License-Identifier: MIT
License: https://opensource.org/license/mit
*)

(*!
<summary>Groups the four cyclic file-content manager scenarios.</summary>
<description>
Owns one independent directory fixture per leaf. Each child borrows and exclusively drives its assigned fixture.
The group keeps the fixtures, Children array and parent associations fixed for the lifetime of the tests.
Use from one task without reentry. Do not copy the group or modify its borrowed Children array.
</description>
*)

{attribute 'no_assign'}
{attribute 'no_explicit_call' := 'do not call this function block directly'}
FUNCTION_BLOCK FileContentManagerOperationsTest EXTENDS TOF_Testing.TestGroup<4>
VAR_STAT
	//! <summary>Class name shared by instances of this concrete function block.</summary>
	{attribute 'hide'}
	_ClassName : STRING := __POUNAME();
END_VAR
VAR
	_TextDirectory : FileTestDirectory(directoryPath := 'C:\OpenFrameworkTests\FileContent_CreateText');
	_ReadOnlyDirectory : FileTestDirectory(directoryPath := 'C:\OpenFrameworkTests\FileContent_ReadOnly');
	_CancelDirectory : FileTestDirectory(directoryPath := 'C:\OpenFrameworkTests\FileContent_Cancel');
	_ReuseDirectory : FileTestDirectory(directoryPath := 'C:\OpenFrameworkTests\FileContent_Reuse');

	_TextTest : FileTextReadWriteTest(
		name := "CreateTextFile",
		parent := THIS^,
		directory := _TextDirectory,
		scenarioTimeout := T#10S
	);
	_ReadOnlyTest : FileReadOnlyWriteTest(
		name := "WriteToFileOpenedForReading",
		parent := THIS^,
		directory := _ReadOnlyDirectory,
		scenarioTimeout := T#15S
	);
	_CancelTest : FileWriteCancellationTest(
		name := "CancelDuringFileWrite",
		parent := THIS^,
		directory := _CancelDirectory,
		scenarioTimeout := T#10S
	);
	_ReuseTest : FileManagerReuseTest(
		name := "ReuseAfterReset",
		parent := THIS^,
		directory := _ReuseDirectory,
		scenarioTimeout := T#20S
	);

	_Children : ARRAY [0.._ChildCount - 1] OF TOF_Testing.ITestElement :=
	[
		_TextTest,
		_ReadOnlyTest,
		_CancelTest,
		_ReuseTest
	];
END_VAR

//! <summary>Borrows the fixed leaf array for this group's lifetime; callers must not modify it.</summary>
{attribute 'monitoring' := 'call'}
PROPERTY Children : REFERENCE TO ARRAY [0.._ChildCount - 1] OF TOF_Testing.ITestElement
GET
Children REF= _Children;
END_GET
END_PROPERTY

//! <summary>Borrows this concrete type name; callers must not modify the referenced storage.</summary>
{attribute 'monitoring' := 'call'}
PROPERTY ClassName : REFERENCE TO STRING
GET
ClassName REF= _ClassName;
END_GET
END_PROPERTY

//! <summary>Borrows the compiler-initialized namespace; callers must not modify the returned reference.</summary>
{attribute 'monitoring' := 'call'}
PROPERTY NamespaceName : REFERENCE TO STRING
GET
NamespaceName REF= CurrentNamespace.Name;
END_GET
END_PROPERTY

//! <summary>Reports this concrete instance size, excluding separately allocated storage.</summary>
{attribute 'monitoring' := 'call'}
PROPERTY SelfSize : ULINT
GET
SelfSize := XSIZEOF(THIS^);
END_GET
END_PROPERTY

END_FUNCTION_BLOCK

// ---- Tests/Files/FileTextReadWriteTest.TcPOU
(*
SPDX-FileCopyrightText: c 2026 Oleksandr Tiutyk <trofimich@gmail.com>
SPDX-License-Identifier: MIT
License: https://opensource.org/license/mit
*)

(*!
<summary>Checks queued text writes, seek and exact readback, followed by string and EOF result guards.</summary>
<description>
Uses a freshly created file inside the owned fixture. Two writes must read back in order.
A separate read past the data establishes a positive EOF result before checking Reset and pre-submission cancellation.
The address check compares buffer identities without reading a result past its documented lifetime.
</description>
*)

{attribute 'no_assign'}
{attribute 'no_explicit_call' := 'do not call this function block directly'}
FUNCTION_BLOCK FileTextReadWriteTest EXTENDS FileContentScenarioTest
VAR_STAT
	//! <summary>Class name shared by instances of this concrete function block.</summary>
	{attribute 'hide'}
	_ClassName : STRING := __POUNAME();
END_VAR
VAR
	_WriteFirst : TOF_FileSystem.WriteString255ToFile(name := "Write first text");
	_WriteSecond : TOF_FileSystem.WriteString255ToFile(name := "Write second text");
	_SeekStart : TOF_FileSystem.SetPositionInFile(name := "Seek to start");
	_ReadText : TOF_FileSystem.ReadString255FromFile(name := "Read text");
	_ReadEof : TOF_FileSystem.ReadString255FromFile(name := "Read after text");
END_VAR

//! <summary>Rearms the borrowed queue children before a new text-file run.</summary>
METHOD PROTECTED ResetScenario : BOOL
ResetScenario := _WriteFirst.Reset()
	AND_THEN _WriteSecond.Reset()
	AND_THEN _SeekStart.Reset()
	AND_THEN _ReadText.Reset()
	AND_THEN _ReadEof.Reset();
END_METHOD

(*!
<summary>Starts or advances the text queue, then verifies read results and their lifetime guards.</summary>
<description>Returns TRUE after all checks pass. The base handles failure reporting and fixture cleanup.</description>
*)
METHOD PROTECTED AdvanceScenario : BOOL
IF _Manager.State.Ready THEN
	_Directory.ExpectFirstFile();
	ConfigureFile(filePath := _Directory.FirstFilePath, modeFlags := _UpdateTextMode);

	_WriteFirst.StringToWrite := 'Test string...';
	_WriteSecond.StringToWrite := 'Another test string...';
	_WriteFirst.Timeout := _NativeTimeout;
	_WriteSecond.Timeout := _NativeTimeout;
	_SeekStart.Position := TOF_Core.SignedInt32.ZERO;
	_SeekStart.Origin := Tc2_System.E_SeekOrigin.SEEK_SET;
	_SeekStart.Timeout := _NativeTimeout;
	_ReadText.Timeout := _NativeTimeout;
	_ReadEof.Timeout := _NativeTimeout;

	_Manager.Enqueue(fileHandleTask := _WriteFirst);
	_Manager.Enqueue(fileHandleTask := _WriteSecond);
	_Manager.Enqueue(fileHandleTask := _SeekStart);
	_Manager.Enqueue(fileHandleTask := _ReadText);
	_Manager.Enqueue(fileHandleTask := _ReadEof);

	IF NOT _Manager.Start() THEN
		_ScenarioFailure := "Prepared text file manager refused Start";
		RETURN;
	END_IF
END_IF

_Manager.Execute();

IF NOT _Manager.State.Stopped THEN
	RETURN;
END_IF

IF NOT _Manager.FinalStopReason.WorkDone THEN
	_ScenarioFailure := "Text file queue did not finish with WorkDone: ";
	TOF_Core.WideStrings.AppendFit(targetString := _ScenarioFailure, sourceString := _Manager.FinalStopReason.Message);
	RETURN;
END_IF

IF _Manager.ResourceManager.ResourceAcquired THEN
	_ScenarioFailure := "File resource remained acquired after the text queue stopped";
	RETURN;
END_IF

AdvanceScenario := checkReadResults();
END_METHOD

(*!
<summary>Checks exact text, a positive EOF, and guarded results after Reset and cancellation.</summary>
<description>Call after all queued operations have stopped and the manager has released its resource.</description>
*)
METHOD PRIVATE checkReadResults : BOOL
VAR
	readAlias : REFERENCE TO STRING(255);
	emptyAlias : REFERENCE TO STRING(255);
END_VAR
IF _ReadText.ReadString <> 'Test string...Another test string...' THEN
	_ScenarioFailure := "Readback did not contain both written strings in order";
	RETURN;
END_IF

IF _ReadEof.ReadString <> '' OR_ELSE NOT _ReadEof.IsEndOfFile THEN
	_ScenarioFailure := "Reading after the written text must return an empty string and EOF";
	RETURN;
END_IF

readAlias REF= _ReadText.ReadString;

IF NOT _ReadText.Reset() OR_ELSE NOT _ReadEof.Reset() THEN
	_ScenarioFailure := "Successful text or EOF read refused Reset";
	RETURN;
END_IF

emptyAlias REF= _ReadText.ReadString;

IF emptyAlias <> '' OR_ELSE _ReadEof.IsEndOfFile THEN
	_ScenarioFailure := "READY read results must expose an empty string and hide previous EOF";
	RETURN;
END_IF

// SA0175: Compare only address identities; the old result contents are no longer borrowed.
{analysis -175}
IF ADR(readAlias) = ADR(emptyAlias) THEN
	_ScenarioFailure := "READY string read must return a separate empty result buffer";
	RETURN;
END_IF
{analysis +175}

IF NOT checkCancelledRead(readTask := _ReadText) THEN
	_ScenarioFailure := "Pre-submission cancellation must hide the old text result";
	RETURN;
END_IF

IF NOT checkCancelledRead(readTask := _ReadEof) THEN
	_ScenarioFailure := "Pre-submission cancellation must hide the old EOF result";
	RETURN;
END_IF

checkReadResults := TRUE;
END_METHOD

(*!
<summary>Verifies cancellation and neutral results for a reset, unbound reader.</summary>
<description>Start and cancel before Execute, with no acquired handle or pending native request.</description>
<param name="readTask">The reset reader from the completed text queue.</param>
*)
METHOD PRIVATE checkCancelledRead : BOOL
VAR_INPUT
	readTask : REFERENCE TO TOF_FileSystem.ReadString255FromFile;
END_VAR
VAR
	cancelAccepted : BOOL;
END_VAR
IF NOT readTask.Start() THEN
	RETURN;
END_IF

cancelAccepted := readTask.Cancel();
readTask.Execute();

checkCancelledRead := cancelAccepted
	AND_THEN readTask.State.Stopped
	AND_THEN readTask.FinalStopReason.ExternalCancel
	AND_THEN readTask.ReadString = ''
	AND_THEN NOT readTask.IsEndOfFile;
END_METHOD

//! <summary>Borrows this concrete type name; callers must not modify the referenced storage.</summary>
{attribute 'monitoring' := 'call'}
PROPERTY ClassName : REFERENCE TO STRING
GET
ClassName REF= _ClassName;
END_GET
END_PROPERTY

//! <summary>Borrows the compiler-initialized namespace; callers must not modify the returned reference.</summary>
{attribute 'monitoring' := 'call'}
PROPERTY NamespaceName : REFERENCE TO STRING
GET
NamespaceName REF= CurrentNamespace.Name;
END_GET
END_PROPERTY

//! <summary>Reports this concrete instance size, excluding separately allocated storage.</summary>
{attribute 'monitoring' := 'call'}
PROPERTY SelfSize : ULINT
GET
SelfSize := XSIZEOF(THIS^);
END_GET
END_PROPERTY

END_FUNCTION_BLOCK

// ---- Tests/Files/FileContentScenarioTest.TcPOU
(*
SPDX-FileCopyrightText: c 2026 Oleksandr Tiutyk <trofimich@gmail.com>
SPDX-License-Identifier: MIT
License: https://opensource.org/license/mit
*)

(*!
<summary>Drives one owned file-content scenario through preparation, execution and cooperative cleanup.</summary>
<description>
The parent owns a distinct directory fixture for this leaf. The leaf exclusively drives that fixture and
its own manager from one task. The scenario deadline includes waiting for the shared root and excludes cleanup.
Derived scenarios advance only one cycle at a time and retain failures in _ScenarioFailure. The leaf reports
after the manager and any independent operations stop and the fixture finishes removal attempts. Native errors can leave
artifacts or a retained resource requiring inspection. Do not copy the leaf or reset the runner while the leaf is active.
</description>
*)

{attribute 'no_assign'}
{attribute 'no_explicit_call' := 'do not call this function block directly'}
FUNCTION_BLOCK ABSTRACT FileContentScenarioTest EXTENDS TOF_Testing.MultiCycleTest
VAR CONSTANT
	//! <summary>Timeout passed to each native file operation.</summary>
	_NativeTimeout : TIME := T#2S;
	//! <summary>Opens a truncated text file for both writing and reading through the same handle.</summary>
	_UpdateTextMode : DWORD := Tc2_System.Global_Variables.FOPEN_MODEWRITE
		OR Tc2_System.Global_Variables.FOPEN_MODEPLUS
		OR Tc2_System.Global_Variables.FOPEN_MODETEXT;
END_VAR
VAR
	_Directory : REFERENCE TO FileTestDirectory;
	_Manager : TOF_FileSystem.FileContentManager(name := "FileContentManager");
	_ScenarioFailure : TOF_Core.ERROR_MESSAGE;

	_ScenarioTimeout : TIME;
	_ScenarioDeadline : Tc2_Standard.TON;
	_Lifecycle : FILE_TEST_LIFECYCLE;
	_CleanupExceptionObserved : BOOL;
END_VAR

(*!
<summary>Borrows the parent-owned fixture and configures the scenario deadline.</summary>
<description>
Performs no I/O. The parent keeps the fixture alive and gives this leaf exclusive use of it.
The inherited initializer stores the display name and parent. The scenario deadline excludes cleanup.
</description>
<param name="name">Name used in the test report.</param>
<param name="parent">Group that owns this leaf and its directory fixture.</param>
<param name="directory">Dedicated fixture with a fixed path inside the shared test root.</param>
<param name="scenarioTimeout">Positive limit for preparation and scenario work.</param>
*)
METHOD FB_init : BOOL
VAR_INPUT
	bInitRetains: BOOL; // TRUE: the retain variables are initialized (reset warm / reset cold)
	bInCopyCode: BOOL; // TRUE: the instance will be copied to the copy code afterward (online change)
	name : WSTRING;
	parent : TOF_Testing.ITestElement;
	directory : REFERENCE TO FileTestDirectory;
	scenarioTimeout : TIME;
END_VAR
IF NOT bInCopyCode THEN
	_Directory REF= directory;
	_ScenarioTimeout := scenarioTimeout;
	// The scenario clock is separate from cleanup, which can span many PLC cycles.
	_Timeout := T#0S;
END_IF

FB_init := TRUE;
END_METHOD

(*!
<summary>Rearms the idle manager, child tasks and directory before a run.</summary>
<description>
A retained resource or unsuccessful fixture cleanup blocks reuse. If preparation for reuse fails, record failure
before any new I/O. Clearing waiting entries also covers a previous Start refusal while the manager was READY.
</description>
*)
METHOD PROTECTED FINAL BeforeTest
IF NOT __ISVALIDREF(_Directory) OR_ELSE _ScenarioTimeout <= T#0S THEN
	RecordFailure(message := "File scenario needs a valid fixture and a positive deadline");
	RETURN;
END_IF

IF _Manager.State.Running OR_ELSE _Manager.ResourceManager.ResourceAcquired OR_ELSE NOT _Manager.Reset() THEN
	RecordFailure(message := "File manager could not be rearmed after the previous run");
	RETURN;
END_IF

_Manager.ClearWaitingTasks();

IF NOT ResetScenario() THEN
	RecordFailure(message := "A file scenario task refused to reset");
	RETURN;
END_IF

IF NOT _Directory.Reset() THEN
	RecordFailure(message := "File scenario directory could not be rearmed; inspect the retained fixture diagnostics");
	RETURN;
END_IF

_ScenarioDeadline(IN := FALSE, PT := _ScenarioTimeout);
_ScenarioFailure := "";
_CleanupExceptionObserved := FALSE;
_Lifecycle := FILE_TEST_LIFECYCLE.RUNNING_SCENARIO;
END_METHOD

(*!
<summary>Rearms the concrete child tasks and restores the scenario's initial step.</summary>
<description>Called with the manager idle and its queue empty. Returns FALSE if a child refuses Reset.</description>
*)
METHOD PROTECTED ABSTRACT ResetScenario : BOOL
END_METHOD

(*!
<summary>Advances one bounded scenario cycle once the test owns its directory.</summary>
<description>
Returns TRUE on successful completion. On failure, use CheckScenario or copy a diagnostic into _ScenarioFailure.
The base waits for stopping and directory cleanup before reporting. Leave any started manager work available
for cooperative cancellation. Override DrainScenario if an independent operation may still be active.
</description>
*)
METHOD PROTECTED ABSTRACT AdvanceScenario : BOOL
END_METHOD

(*!
<summary>Retains the first failed condition for reporting after cooperative cleanup.</summary>
<description>
Use during AdvanceScenario. This never marks the test finished or interrupts the current callback.
The base starts cleanup after the callback returns.
</description>
<param name="condition">Condition required for the scenario to pass.</param>
<param name="message">Nonempty diagnostic for a false condition.</param>
*)
METHOD PROTECTED FINAL CheckScenario
VAR_INPUT
	condition : BOOL;
	message : WSTRING(255);
END_VAR
IF NOT condition AND_THEN _ScenarioFailure = "" THEN
	_ScenarioFailure := message;
END_IF
END_METHOD

(*!
<summary>Advances stopping of any operations driven independently from the file manager.</summary>
<description>
Called after the manager stops and before the fixture attempts removal. Override only if the scenario starts
operations outside the manager. Return FALSE while any such operation still needs cyclic work.
The default returns TRUE. An exception delays cleanup for retry and is recorded as a cleanup failure.
</description>
*)
METHOD PROTECTED DrainScenario : BOOL
DrainScenario := TRUE;
END_METHOD

(*!
<summary>Configures the idle manager to open an owned fixture file using the specified access and format.</summary>
<description>Call before Start. The queue stops when its last operation finishes.</description>
<param name="filePath">Absolute path of the registered file inside this scenario's directory.</param>
<param name="modeFlags">Beckhoff file-open access and format flags.</param>
*)
METHOD PROTECTED FINAL ConfigureFile
VAR_INPUT
	filePath : Tc2_System.T_MaxString;
	modeFlags : DWORD;
END_VAR
_Manager.FilePath := filePath;
_Manager.ModeFlags := modeFlags;
_Manager.PathType := Tc2_System.E_OpenPath.PATH_GENERIC;
_Manager.Timeout := _NativeTimeout;
_Manager.StopWhenNoPendingTasks := TRUE;
END_METHOD

(*!
<summary>Advances file work or cooperative cleanup and publishes the resulting outcome.</summary>
<description>
A scenario exception enters the same cleanup phase as an ordinary failure. The manager and independent operations
are drained before fixture removal. A cleanup interruption is retained and retried on later calls.
The inherited test boundary handles the terminal allocation latch.
</description>
*)
METHOD PROTECTED FINAL ExecuteTest : TOF_Testing.TEST_CYCLE_RESULT
VAR
	exceptionCode : __SYSTEM.ExceptionCode;
	exception : TOF_Core.IException;
	finished : BOOL;
	scenarioDiagnostic : TOF_Core.ERROR_MESSAGE;
	cleanupFailure : TOF_Core.ERROR_MESSAGE;
END_VAR
ExecuteTest := TOF_Testing.TEST_CYCLE_RESULT.BUSY;

IF _Lifecycle = FILE_TEST_LIFECYCLE.RUNNING_SCENARIO THEN
	__TRY
		finished := runScenario();
	__CATCH(exceptionCode)
		IF _ScenarioFailure = "" THEN
			_ScenarioFailure := "Exception interrupted fixture preparation or file work";

			__TRY
				exception := TOF_Core.ExceptionManager.GetLastException(
					exceptionCode := exceptionCode,
					catchPointNamespaceName := NamespaceName,
					catchPointPOUName := __POUNAME(),
					catchPointPosition := __POSITION()
				);

				IF exception <> 0 THEN
					scenarioDiagnostic := exception.GetMessage();

					IF scenarioDiagnostic <> "" THEN
						_ScenarioFailure := scenarioDiagnostic;
					END_IF
				END_IF
			__CATCH
				(* Preserve the copied fallback if diagnostic formatting fails. *)
			__ENDTRY
		END_IF
	__ENDTRY

	IF finished OR_ELSE _ScenarioFailure <> "" THEN
		_Lifecycle := FILE_TEST_LIFECYCLE.CLEANING_UP;
	END_IF

	RETURN;
END_IF

__TRY
	IF _Manager.State.Running THEN
		_Manager.Cancel();
		_Manager.Execute();

		IF _Manager.State.Running THEN
			RETURN;
		END_IF
	END_IF

	IF NOT DrainScenario() THEN
		RETURN;
	END_IF

	_Directory.Cleanup();
__CATCH
	_CleanupExceptionObserved := TRUE;
	RETURN;
__ENDTRY

IF NOT _Directory.CleanupComplete THEN
	RETURN;
END_IF

IF NOT _Directory.CleanupSucceeded OR_ELSE _Directory.CleanupMessage <> TOF_Core.Strings.Empty THEN
	cleanupFailure := TOF_Core.WideStrings.ConcatFit255(
		"Directory cleanup reported a problem for ",
		TO_WSTRING(_Directory.DirectoryPath),
		": ",
		TO_WSTRING(_Directory.CleanupMessage)
	);
ELSIF _Manager.ResourceManager.ResourceAcquired THEN
	cleanupFailure := "File manager still reports an acquired resource after stopping";
ELSIF _CleanupExceptionObserved THEN
	cleanupFailure := "An exception interrupted a cleanup attempt";
END_IF

IF cleanupFailure <> "" THEN
	IF _ScenarioFailure <> "" THEN
		TOF_Core.WideStrings.AppendFit(targetString := _ScenarioFailure, sourceString := " | ");
	END_IF

	TOF_Core.WideStrings.AppendFit(targetString := _ScenarioFailure, sourceString := cleanupFailure);
END_IF

_Lifecycle := FILE_TEST_LIFECYCLE.FINISHED;
ExecuteTest := TOF_Testing.TEST_CYCLE_RESULT.DONE;

IF _ScenarioFailure <> "" THEN
	RecordFailure(message := _ScenarioFailure);
END_IF
END_METHOD

(*!
<summary>Prepares the owned directory and dispatches one bounded scenario cycle.</summary>
<description>
The deadline applies even while waiting for the shared root. Returns the scenario completion signal.
Retains deployment, ownership or deadline failures for reporting after cleanup.
</description>
*)
METHOD PRIVATE runScenario : BOOL
_ScenarioDeadline(IN := TRUE, PT := _ScenarioTimeout);

IF FileTestRoot.FailureMessage <> TOF_Core.Strings.Empty THEN
	_ScenarioFailure := TO_WSTRING(FileTestRoot.FailureMessage);
	RETURN;
END_IF

IF _ScenarioDeadline.Q THEN
	IF NOT FileTestRoot.Prepared THEN
		_ScenarioFailure := "Shared filesystem test root was not ready before the scenario deadline";
	ELSIF NOT _Directory.Prepared THEN
		_ScenarioFailure := "Scenario directory preparation exceeded its deadline";
	ELSE
		_ScenarioFailure := "File work exceeded the scenario deadline";
	END_IF

	RETURN;
END_IF

IF NOT FileTestRoot.Prepared THEN
	RETURN;
END_IF

IF NOT _Directory.Prepared THEN
	_Directory.Prepare();

	IF _Directory.PreparationFailed THEN
		_ScenarioFailure := TOF_Core.WideStrings.ConcatFit255(
			TO_WSTRING(_Directory.DirectoryPath), ": ", TO_WSTRING(_Directory.PreparationMessage)
		);
		RETURN;
	END_IF

	IF NOT _Directory.Prepared THEN
		RETURN;
	END_IF
END_IF

runScenario := AdvanceScenario();
END_METHOD

END_FUNCTION_BLOCK

// ---- Tests/Files/FileReadOnlyWriteTest.TcPOU
(*
SPDX-FileCopyrightText: c 2026 Oleksandr Tiutyk <trofimich@gmail.com>
SPDX-License-Identifier: MIT
License: https://opensource.org/license/mit
*)

(*!
<summary>Checks native write failure on a read-only text handle and propagation through the file queue.</summary>
<description>
Creates and releases an empty file first, then reopens it for reading and queues a write followed by a read.
The native write error must reach the manager and leave the successor unstarted.
</description>
*)

{attribute 'no_assign'}
{attribute 'no_explicit_call' := 'do not call this function block directly'}
FUNCTION_BLOCK FileReadOnlyWriteTest EXTENDS FileContentScenarioTest
VAR_STAT
	//! <summary>Class name shared by instances of this concrete function block.</summary>
	{attribute 'hide'}
	_ClassName : STRING := __POUNAME();
END_VAR
VAR
	_Step : READ_ONLY_FILE_TEST_STEP;
	_WriteText : TOF_FileSystem.WriteString255ToFile(name := "Write through read-only handle");
	_WaitingRead : TOF_FileSystem.ReadString255FromFile(name := "Read after failed write");
END_VAR

//! <summary>Restores empty-file preparation and resets both child operations for reuse.</summary>
METHOD PROTECTED ResetScenario : BOOL
_Step := READ_ONLY_FILE_TEST_STEP.CREATE_FILE;
ResetScenario := _WriteText.Reset() AND_THEN _WaitingRead.Reset();
END_METHOD

(*!
<summary>Creates the input file, opens it read-only and advances the failing queue.</summary>
<description>Returns TRUE once the write diagnostic reached the manager and the successor stayed READY.</description>
*)
METHOD PROTECTED AdvanceScenario : BOOL
VAR
	writeMessage : WSTRING(255);
END_VAR
CASE _Step OF
	READ_ONLY_FILE_TEST_STEP.CREATE_FILE:
		_Directory.ExpectFirstFile();
		ConfigureFile(
			filePath := _Directory.FirstFilePath,
			modeFlags := Tc2_System.Global_Variables.FOPEN_MODEWRITE OR Tc2_System.Global_Variables.FOPEN_MODETEXT
		);

		IF NOT _Manager.Start() THEN
			_ScenarioFailure := "Empty file preparation refused Start";
			RETURN;
		END_IF

		_Step := READ_ONLY_FILE_TEST_STEP.OPEN_FILE_FOR_READING;

	READ_ONLY_FILE_TEST_STEP.OPEN_FILE_FOR_READING:
		_Manager.Execute();

		IF NOT _Manager.State.Stopped THEN
			RETURN;
		END_IF

		IF NOT _Manager.FinalStopReason.WorkDone OR_ELSE _Manager.ResourceManager.ResourceAcquired THEN
			_ScenarioFailure := "Fixture creation must succeed and release the file before reopening it";
			RETURN;
		END_IF

		IF NOT _Manager.Reset() THEN
			_ScenarioFailure := "File manager refused Reset before reopening the fixture for reading";
			RETURN;
		END_IF

		ConfigureFile(
			filePath := _Directory.FirstFilePath,
			modeFlags := Tc2_System.Global_Variables.FOPEN_MODEREAD OR Tc2_System.Global_Variables.FOPEN_MODETEXT
		);
		_WriteText.StringToWrite := 'This text must be rejected by the read-only handle';
		_WriteText.Timeout := _NativeTimeout;
		_Manager.Enqueue(fileHandleTask := _WriteText);
		_Manager.Enqueue(fileHandleTask := _WaitingRead);

		IF NOT _Manager.Start() THEN
			_ScenarioFailure := "Prepared read-only file manager refused Start before executing the write";
			RETURN;
		END_IF

		_Step := READ_ONLY_FILE_TEST_STEP.CHECK_WRITE_FAILURE;

	READ_ONLY_FILE_TEST_STEP.CHECK_WRITE_FAILURE:
		_Manager.Execute();

		IF NOT _Manager.State.Stopped THEN
			RETURN;
		END_IF

		writeMessage := _WriteText.FinalStopReason.Message;

		IF NOT _WriteText.State.Stopped OR_ELSE NOT _WriteText.FinalStopReason.Failure THEN
			_ScenarioFailure := "The write child must fail on a handle opened for reading";
		ELSIF NOT TOF_Core.WideStrings.Contains(
			stringToSearchIn := writeMessage,
			stringToFind := "writing string to file"
		)
		THEN
			_ScenarioFailure := "The write child failed without the native string-write diagnostic";
		ELSIF NOT _Manager.FinalStopReason.Failure THEN
			_ScenarioFailure := "File manager must stop with Failure after a failed write";
		ELSIF _Manager.FinalStopReason.Message <> _WriteText.FinalStopReason.Message THEN
			_ScenarioFailure := "File manager must preserve the failed child's diagnostic";
		ELSIF NOT _WaitingRead.State.Ready THEN
			_ScenarioFailure := "The read queued after the failed write must remain READY";
		ELSE
			AdvanceScenario := TRUE;
		END_IF
END_CASE
END_METHOD

//! <summary>Borrows this concrete type name; callers must not modify the referenced storage.</summary>
{attribute 'monitoring' := 'call'}
PROPERTY ClassName : REFERENCE TO STRING
GET
ClassName REF= _ClassName;
END_GET
END_PROPERTY

//! <summary>Borrows the compiler-initialized namespace; callers must not modify the returned reference.</summary>
{attribute 'monitoring' := 'call'}
PROPERTY NamespaceName : REFERENCE TO STRING
GET
NamespaceName REF= CurrentNamespace.Name;
END_GET
END_PROPERTY

//! <summary>Reports this concrete instance size, excluding separately allocated storage.</summary>
{attribute 'monitoring' := 'call'}
PROPERTY SelfSize : ULINT
GET
SelfSize := XSIZEOF(THIS^);
END_GET
END_PROPERTY

END_FUNCTION_BLOCK

// ---- Tests/Files/FileWriteCancellationTest.TcPOU
(*
SPDX-FileCopyrightText: c 2026 Oleksandr Tiutyk <trofimich@gmail.com>
SPDX-License-Identifier: MIT
License: https://opensource.org/license/mit
*)

(*!
<summary>Checks cancellation of a pending native write before its queued successor can execute.</summary>
<description>
Requires an observed busy native write and an accepted Cancel request. The manager must retain the handle
until the active child finishes stopping, then release it and leave the queued read unstarted.
A write that finishes before its busy state is observed fails this scenario.
</description>
*)

{attribute 'no_assign'}
{attribute 'no_explicit_call' := 'do not call this function block directly'}
FUNCTION_BLOCK FileWriteCancellationTest EXTENDS FileContentScenarioTest
VAR_STAT
	//! <summary>Class name shared by instances of this concrete function block.</summary>
	{attribute 'hide'}
	_ClassName : STRING := __POUNAME();
END_VAR
VAR
	_WriteText : TOF_FileSystem.WriteString255ToFile(name := "Cancel active text write");
	_WaitingRead : TOF_FileSystem.ReadString255FromFile(name := "Read after cancelled write");
	_CancelRequested : BOOL;
END_VAR

//! <summary>Clears the cancellation observation and rearms both queue children.</summary>
METHOD PROTECTED ResetScenario : BOOL
_CancelRequested := FALSE;
ResetScenario := _WriteText.Reset() AND_THEN _WaitingRead.Reset();
END_METHOD

(*!
<summary>Starts the queue and requests cancellation only after observing native write activity.</summary>
<description>Returns TRUE on verified cancellation. The base reports cleanup and retained failures.</description>
*)
METHOD PROTECTED AdvanceScenario : BOOL
IF _Manager.State.Ready THEN
	_Directory.ExpectFirstFile();
	ConfigureFile(filePath := _Directory.FirstFilePath, modeFlags := _UpdateTextMode);

	_WriteText.StringToWrite := 'Cancel while the native file write is pending';
	_WriteText.Timeout := _NativeTimeout;
	_WaitingRead.Timeout := _NativeTimeout;
	_Manager.Enqueue(fileHandleTask := _WriteText);
	_Manager.Enqueue(fileHandleTask := _WaitingRead);

	IF NOT _Manager.Start() THEN
		_ScenarioFailure := "File manager refused Start before the cancellation check";
		RETURN;
	END_IF
END_IF

_Manager.Execute();

IF _WriteText.FileOperationInProgress THEN
	IF NOT _Manager.ResourceManager.ResourceAcquired THEN
		_ScenarioFailure := "The file resource must remain acquired while its write is busy";
		RETURN;
	END_IF

	IF NOT _CancelRequested THEN
		_CancelRequested := _Manager.Cancel();

		IF NOT _CancelRequested THEN
			_ScenarioFailure := "File manager must accept Cancel during a pending native write";
			RETURN;
		END_IF
	END_IF
END_IF

IF _Manager.RunningSubstate.ResourceReleasing AND_THEN NOT _WriteText.State.Stopped THEN
	_ScenarioFailure := "File resource release began before the active write child stopped";
	RETURN;
END_IF

IF NOT _CancelRequested AND_THEN (_WriteText.State.Stopped OR_ELSE _Manager.State.Stopped) THEN
	_ScenarioFailure := "Write or manager stopped before the test observed a busy native write and requested Cancel";
	RETURN;
END_IF

IF NOT _Manager.State.Stopped THEN
	RETURN;
END_IF

IF NOT _Manager.FinalStopReason.ExternalCancel THEN
	_ScenarioFailure := "File manager must stop with ExternalCancel";
ELSIF NOT _WriteText.State.Stopped OR_ELSE NOT _WriteText.FinalStopReason.ExternalCancel THEN
	_ScenarioFailure := "The active write must stop with ExternalCancel";
ELSIF _WriteText.FileOperationInProgress THEN
	_ScenarioFailure := "The native write must no longer be busy after the manager stops";
ELSIF NOT _WaitingRead.State.Ready THEN
	_ScenarioFailure := "The read queued after the cancelled write must remain READY";
ELSE
	AdvanceScenario := TRUE;
END_IF
END_METHOD

//! <summary>Borrows this concrete type name; callers must not modify the referenced storage.</summary>
{attribute 'monitoring' := 'call'}
PROPERTY ClassName : REFERENCE TO STRING
GET
ClassName REF= _ClassName;
END_GET
END_PROPERTY

//! <summary>Borrows the compiler-initialized namespace; callers must not modify the returned reference.</summary>
{attribute 'monitoring' := 'call'}
PROPERTY NamespaceName : REFERENCE TO STRING
GET
NamespaceName REF= CurrentNamespace.Name;
END_GET
END_PROPERTY

//! <summary>Reports this concrete instance size, excluding separately allocated storage.</summary>
{attribute 'monitoring' := 'call'}
PROPERTY SelfSize : ULINT
GET
SelfSize := XSIZEOF(THIS^);
END_GET
END_PROPERTY

END_FUNCTION_BLOCK

// ---- Tests/Files/FileManagerReuseTest.TcPOU
(*
SPDX-FileCopyrightText: c 2026 Oleksandr Tiutyk <trofimich@gmail.com>
SPDX-License-Identifier: MIT
License: https://opensource.org/license/mit
*)

(*!
<summary>Checks manager Reset and child reuse after cancellation between queued file operations.</summary>
<description>
The first write succeeds and one read remains queued when the manager stops. Reset must remove that
entry and clear the file path. The second queue uses the same manager and write task on a different file.
It must read back the second text and leave the removed read unstarted.
</description>
*)

{attribute 'no_assign'}
{attribute 'no_explicit_call' := 'do not call this function block directly'}
FUNCTION_BLOCK FileManagerReuseTest EXTENDS FileContentScenarioTest
VAR_STAT
	//! <summary>Class name shared by instances of this concrete function block.</summary>
	{attribute 'hide'}
	_ClassName : STRING := __POUNAME();
END_VAR
VAR CONSTANT
	//! <summary>Text written and expected back exclusively in the second run.</summary>
	_SecondFileText : STRING := 'FileContentManager reused after Reset';
END_VAR
VAR
	_Step : FILE_MANAGER_REUSE_TEST_STEP;
	_WriteText : TOF_FileSystem.WriteString255ToFile(name := "Write on each run");
	_WaitingRead : TOF_FileSystem.ReadString255FromFile(name := "Read removed by Reset");
	_SeekStart : TOF_FileSystem.SetPositionInFile(name := "Seek on second run");
	_ReadText : TOF_FileSystem.ReadString255FromFile(name := "Read on second run");
END_VAR

//! <summary>Restores the first-run phase and rearms the children for a new test-runner pass.</summary>
METHOD PROTECTED ResetScenario : BOOL
_Step := FILE_MANAGER_REUSE_TEST_STEP.START_FIRST_WRITE;
ResetScenario := _WriteText.Reset()
	AND_THEN _WaitingRead.Reset()
	AND_THEN _SeekStart.Reset()
	AND_THEN _ReadText.Reset();
END_METHOD

(*!
<summary>Advances the cancelled first queue and the reconfigured second queue.</summary>
<description>Returns TRUE after the exact second readback and the unused successor have been verified.</description>
*)
METHOD PROTECTED AdvanceScenario : BOOL
CASE _Step OF
	FILE_MANAGER_REUSE_TEST_STEP.START_FIRST_WRITE:
		_Directory.ExpectFirstFile();
		ConfigureFile(filePath := _Directory.FirstFilePath, modeFlags := _UpdateTextMode);

		_WriteText.StringToWrite := 'First run before Reset';
		_WriteText.Timeout := _NativeTimeout;
		_WaitingRead.Timeout := _NativeTimeout;
		_SeekStart.Timeout := _NativeTimeout;
		_ReadText.Timeout := _NativeTimeout;
		_Manager.Enqueue(fileHandleTask := _WriteText);
		_Manager.Enqueue(fileHandleTask := _WaitingRead);

		IF NOT _Manager.Start() THEN
			_ScenarioFailure := "File manager refused Start before the first write";
			RETURN;
		END_IF

		_Step := FILE_MANAGER_REUSE_TEST_STEP.CANCEL_AFTER_WRITE;

	FILE_MANAGER_REUSE_TEST_STEP.CANCEL_AFTER_WRITE:
		_Manager.Execute();

		IF _Manager.State.Stopped THEN
			_ScenarioFailure := "First queue stopped before cancellation between tasks";
			RETURN;
		END_IF

		IF _WriteText.State.Stopped THEN
			IF NOT _WriteText.FinalStopReason.WorkDone OR_ELSE NOT _WaitingRead.State.Ready THEN
				_ScenarioFailure := "First write must finish with WorkDone while its successor is still READY";
				RETURN;
			END_IF

			IF NOT _Manager.Cancel() THEN
				_ScenarioFailure := "File manager refused Cancel between the completed write and the waiting read";
				RETURN;
			END_IF

			_Step := FILE_MANAGER_REUSE_TEST_STEP.RESET_AND_START_SECOND_FILE;
		END_IF

	FILE_MANAGER_REUSE_TEST_STEP.RESET_AND_START_SECOND_FILE:
		_Manager.Execute();

		IF _Manager.State.Stopped AND_THEN resetAndStartSecondFile() THEN
			_Step := FILE_MANAGER_REUSE_TEST_STEP.CHECK_SECOND_FILE;
		END_IF

	FILE_MANAGER_REUSE_TEST_STEP.CHECK_SECOND_FILE:
		_Manager.Execute();

		IF NOT _Manager.State.Stopped THEN
			RETURN;
		END_IF

		IF NOT _Manager.FinalStopReason.WorkDone THEN
			_ScenarioFailure := "Second queue did not finish with WorkDone: ";
			TOF_Core.WideStrings.AppendFit(
				targetString := _ScenarioFailure,
				sourceString := _Manager.FinalStopReason.Message
			);
		ELSIF _ReadText.ReadString <> _SecondFileText THEN
			_ScenarioFailure := "Second queue did not read back the new text written after Reset";
		ELSIF NOT _WaitingRead.State.Ready THEN
			_ScenarioFailure := "The waiting read removed by Reset ran during the second queue";
		ELSE
			AdvanceScenario := TRUE;
		END_IF
END_CASE
END_METHOD

(*!
<summary>Verifies cancellation and Reset before configuring the same manager and write task for the second file.</summary>
<description>Called when the first queue is STOPPED. Returns TRUE only after the second queue accepts Start.</description>
*)
METHOD PRIVATE resetAndStartSecondFile : BOOL
IF NOT _Manager.FinalStopReason.ExternalCancel OR_ELSE _Manager.ResourceManager.ResourceAcquired THEN
	_ScenarioFailure := "First queue must finish with ExternalCancel and release its file before Reset";
	RETURN;
END_IF

IF _Manager.PendingTaskCount <> 1 OR_ELSE NOT _WaitingRead.State.Ready THEN
	_ScenarioFailure := "Exactly one READY read must remain in the queue before Reset";
	RETURN;
END_IF

IF NOT _Manager.Reset() THEN
	_ScenarioFailure := "Stopped file manager refused Reset before the second run";
	RETURN;
END_IF

IF NOT _Manager.State.Ready OR_ELSE _Manager.PendingTaskCount <> 0 OR_ELSE _Manager.FilePath <> '' THEN
	_ScenarioFailure := "Reset must return the file manager to READY, clear its queue and clear its path";
	RETURN;
END_IF

IF NOT _WriteText.Reset() THEN
	_ScenarioFailure := "Completed write refused Reset before reuse";
	RETURN;
END_IF

_Directory.ExpectSecondFile();
ConfigureFile(filePath := _Directory.SecondFilePath, modeFlags := _UpdateTextMode);
_WriteText.StringToWrite := _SecondFileText;
_SeekStart.Position := TOF_Core.SignedInt32.ZERO;
_SeekStart.Origin := Tc2_System.E_SeekOrigin.SEEK_SET;
_Manager.Enqueue(fileHandleTask := _WriteText);
_Manager.Enqueue(fileHandleTask := _SeekStart);
_Manager.Enqueue(fileHandleTask := _ReadText);

resetAndStartSecondFile := _Manager.Start();

IF NOT resetAndStartSecondFile THEN
	_ScenarioFailure := "File manager refused Start for the reconfigured second queue";
END_IF
END_METHOD

//! <summary>Borrows this concrete type name; callers must not modify the referenced storage.</summary>
{attribute 'monitoring' := 'call'}
PROPERTY ClassName : REFERENCE TO STRING
GET
ClassName REF= _ClassName;
END_GET
END_PROPERTY

//! <summary>Borrows the compiler-initialized namespace; callers must not modify the returned reference.</summary>
{attribute 'monitoring' := 'call'}
PROPERTY NamespaceName : REFERENCE TO STRING
GET
NamespaceName REF= CurrentNamespace.Name;
END_GET
END_PROPERTY

//! <summary>Reports this concrete instance size, excluding separately allocated storage.</summary>
{attribute 'monitoring' := 'call'}
PROPERTY SelfSize : ULINT
GET
SelfSize := XSIZEOF(THIS^);
END_GET
END_PROPERTY

END_FUNCTION_BLOCK

// ---- Tests/Files/FileSystemIntegrationTestGroup.TcPOU
(*
SPDX-FileCopyrightText: © 2026 Oleksandr Tiutyk <trofimich@gmail.com>
SPDX-License-Identifier: MIT
License: https://opensource.org/license/mit
*)

(*!
<summary>Groups the native byte, buffer validation and caller-exception filesystem integration cases.</summary>
<description>
Owns an independent directory fixture per leaf. Each child borrows and exclusively drives its assigned fixture.
The group and its fixed child array have the same lifetime. Use from one task and do not copy the group.
</description>
*)

{attribute 'no_assign'}
{attribute 'no_explicit_call' := 'do not call this function block directly'}
FUNCTION_BLOCK FileSystemIntegrationTestGroup EXTENDS TOF_Testing.TestGroup<3>
VAR_STAT
	//! <summary>Class name shared by instances of this concrete function block.</summary>
	{attribute 'hide'}
	_ClassName : STRING := __POUNAME();
END_VAR
VAR
	_OperationsDirectory : FileTestDirectory(directoryPath := 'C:\OpenFrameworkTests\FileSystem_Operations');
	_BuffersDirectory : FileTestDirectory(directoryPath := 'C:\OpenFrameworkTests\FileSystem_Buffers');
	_CallerDirectory : FileTestDirectory(directoryPath := 'C:\OpenFrameworkTests\FileSystem_CallerException');

	_ByteOperations : FileByteOperationsTest(
		name := "ByteFileOperationsAndGuards",
		parent := THIS^,
		directory := _OperationsDirectory,
		scenarioTimeout := T#30S
	);
	_BufferMatrix : FileBinaryBufferMatrixTest(
		name := "BinaryBufferMatrix",
		parent := THIS^,
		directory := _BuffersDirectory,
		scenarioTimeout := T#30S
	);
	_CallerCleanup : FileCallerExceptionCleanupTest(
		name := "CaughtCallerExceptionCleanup",
		parent := THIS^,
		directory := _CallerDirectory,
		scenarioTimeout := T#15S
	);

	_Children : ARRAY [0.._ChildCount - 1] OF TOF_Testing.ITestElement :=
		[_ByteOperations, _BufferMatrix, _CallerCleanup];
END_VAR

//! <summary>Borrows the fixed leaf array for this group; callers must not modify it.</summary>
{attribute 'monitoring' := 'call'}
PROPERTY Children : REFERENCE TO ARRAY [0.._ChildCount - 1] OF TOF_Testing.ITestElement
GET
Children REF= _Children;
END_GET
END_PROPERTY

//! <summary>Borrows the concrete type name; callers must not modify the referenced storage.</summary>
{attribute 'monitoring' := 'call'}
PROPERTY ClassName : REFERENCE TO STRING
GET
ClassName REF= _ClassName;
END_GET
END_PROPERTY

//! <summary>Borrows the compiler-initialized namespace; callers must not modify it.</summary>
{attribute 'monitoring' := 'call'}
PROPERTY NamespaceName : REFERENCE TO STRING
GET
NamespaceName REF= CurrentNamespace.Name;
END_GET
END_PROPERTY

